ACTION ErrorHandling:
// Alarm_0280	280	Error	Błąd czujnika temperatury zbiornika
// Alarm_0281	281	Error	Błąd grzania zbiornika, brak wzrostu temperatury

IF bAlarmInit THEN
    bAlarmInit := FALSE; 
	fbSourceInfo.Clear();
	fbSourceInfo.sName:=wsLiteral_TO_UTF8(sStationName);//'Machine';
	fbSourceInfo.nId:=iStationIndex;//2700;
	// Alarm_0280	280	Error	Błąd czujnika temperatury zbiornika
    arfbAlarm[0].CreateEx(stEventEntry := TC_EVENTS.AlarmClass.Alarm_0280, bWithConfirmation:= FALSE,  ipSourceInfo:= fbSourceInfo); 
	// Alarm_0281	281	Error	Błąd grzania zbiornika, brak wzrostu temperatury
	arfbAlarm[1].CreateEx(stEventEntry := TC_EVENTS.AlarmClass.Alarm_0281, bWithConfirmation:= FALSE,  ipSourceInfo:= fbSourceInfo);
END_IF
	

//************LISTA BŁĘDÓW***************
bStateError:= (eState=E_Station.eError) OR (eState=E_Station.eResetting) OR bIgnoreError;

IF bEnable THEN
	// Alarm_0280	280	Error	Błąd czujnika temperatury zbiornika
	//Error 1 - Błąd czujnika temperatury zbiornika
	IF (bTemperatureSensorFault OR lrHeaterTemperatureCVSensor = 0 ) THEN
		IF NOT arfbAlarm[0].bActive THEN
			bTempRegulatorReset 	:= TRUE;
			arfbAlarm[0].Raise(nTimeStamp:=0);
		END_IF
	ELSE	
		IF  arfbAlarm[0].bActive AND bReset THEN
			arfbAlarm[0].Clear(nTimeStamp:=0, bResetConfirmation:= FALSE);
		END_IF
// 		bTempRegulatorReset 	:= TRUE;
// 		bError := TRUE;
// 		nErrorNr 				:= 181;
// 		//nErrorNr				:=nErrorNr+iStationIndex;
// 		sErrorDescription 		:= 'Błąd czujnika temperatury zbiornika';	
	END_IF
	// Alarm_0281	281	Error	Błąd grzania zbiornika, brak wzrostu temperatury
	//Error 2 - Błąd czujnika temperatury
	tofbHeaterPWMOut(IN:=bHeaterPWMOut,PT:=T#30S);
	tonHeaterOnAndNotHeating(IN:=tofbHeaterPWMOut.Q AND lrHeaterTemperatureCVSensor=lrHeaterTemperatureCVSensorLast AND NOT bIgnoreError , PT:=T#5M);
	lrHeaterTemperatureCVSensorLast := lrHeaterTemperatureCVSensor;
	IF tonHeaterOnAndNotHeating.Q THEN
		IF NOT arfbAlarm[1].bActive THEN
			bTempRegulatorReset 	:= TRUE;
			arfbAlarm[1].Raise(nTimeStamp:=0);
		END_IF
	ELSE	
		IF  arfbAlarm[1].bActive AND bReset THEN
			arfbAlarm[1].Clear(nTimeStamp:=0, bResetConfirmation:= FALSE);
		END_IF
//  		bTempRegulatorReset 	:= TRUE;
// 		bError := TRUE;
// 		nErrorNr 				:= 182;
// 		//nErrorNr				:=nErrorNr+iStationIndex;
// 		sErrorDescription 		:= 'Błąd grzania zbiornika, brak wzrostu temperatury';	
	END_IF
ELSE
		bError := FALSE;
END_IF
//*******KONIEC LISTA BŁĘDÓW***************

IF bError AND NOT bStateError THEN
	IF eLastState = eRunning THEN
		bCycleNotDone := TRUE;
	END_IF
	eState := E_Station.eError;
END_IF

(*Wyświetlanie błedu na wyjściu*)
bError							:= FALSE;
FOR nAlarmNumerator := 0 TO 19 DO
	bError						:= bError OR arfbAlarm[nAlarmNumerator].bActive;
END_FOR

(*Przepisywanie nazwy stacji*)
sErrorStationName:=WSTRING_TO_STRING(sStationName);
END_ACTION

ACTION HeaterRegulator:
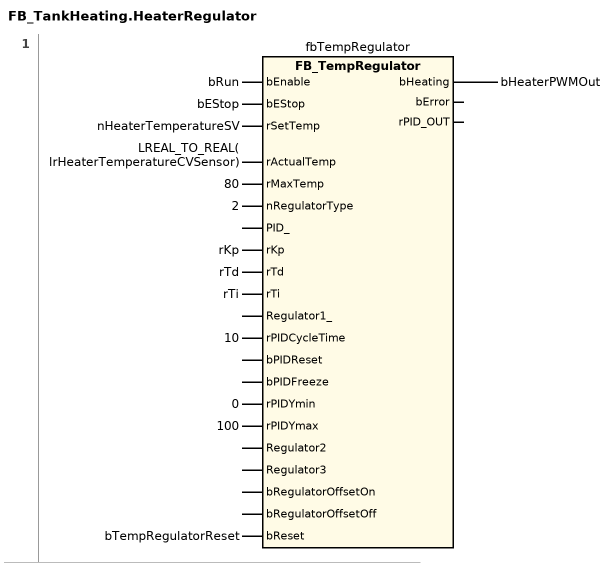
// NETWORK 1
fbTempRegulator(
    bEnable := bRun,
    bEStop := bEStop,
    rSetTemp := nHeaterTemperatureSV,
    rActualTemp := LREAL_TO_REAL(lrHeaterTemperatureCVSensor),
    rMaxTemp := 80,
    nRegulatorType := 2,
    rKp := rKp,
    rTd := rTd,
    rTi := rTi,
    rPIDCycleTime := 10,
    rPIDYmin := 0,
    rPIDYmax := 100,
    bReset := bTempRegulatorReset); // FB_TempRegulator
bHeaterPWMOut := fbTempRegulator.bHeating;
END_ACTION

ACTION Running:

CASE eRunningState OF
	/////////////////////////////	
	E_MassHeatingState.eDisabled:		//Wyłączona
		
		IF bRun THEN
			eRunningState := E_MassHeatingState.eHeating;
		END_IF
		
	/////////////////////////////	
	E_MassHeatingState.eHeating:		//Grzanie
	
		IF (ABS(lrHeaterTemperatureCVSensor-nHeaterTemperatureSV)<nTempHisteresis OR bIgnoreError) THEN
			eRunningState:=E_MassHeatingState.eReady;	
		END_IF
		IF NOT bRun THEN
			eRunningState := E_MassHeatingState.eCooling;
		END_IF
	
	/////////////////////////////	
	E_MassHeatingState.eReady:			//Gotowość
	
		IF (ABS(lrHeaterTemperatureCVSensor-nHeaterTemperatureSV)>nTempHisteresis AND NOT bIgnoreError) THEN
			eRunningState:=E_MassHeatingState.eHeating;
		END_IF
		IF NOT bRun THEN
			eRunningState := E_MassHeatingState.eCooling;
		END_IF
	
	/////////////////////////////	
	E_MassHeatingState.eCooling:		//Chłodzenie
		IF lrHeaterTemperatureCVSensor < 40 THEN
			eRunningState := E_MassHeatingState.eDisabled;
		END_IF
		IF bRun THEN
			eRunningState := E_MassHeatingState.eHeating;
		END_IF

END_CASE
END_ACTION

END_FUNCTION_BLOCK

// ---- POUs/FB/FB_WriteDataToArrayString.TcPOU
FUNCTION_BLOCK FB_WriteDataToArrayString
VAR_INPUT
	bWrite:BOOL;
	nCycleTime:INT;
	lrData1:LREAL;
	lrData2:LREAL;
	lrData2B:LREAL;
	bData3:BOOL;
	bData4:BOOL;
	bData5:BOOL;
	bData2B_ON:BOOL;
END_VAR
VAR_OUTPUT
	AsData:ARRAY [0..500] OF STRING;
END_VAR
VAR
	i: INT;
	sTemp1: STRING;
	sTemp2: STRING;
	sTemp3: STRING;
	sTemp4: STRING;
	sTemp5: STRING;	
	sTemp6: STRING;
	sTemp7: STRING;
	sTemp8: STRING;
	sTemp9: STRING;	
	sTemp10: STRING;	
	sTemp11: STRING;	
	sTemp12: STRING;
	sTemp13: STRING;	
	rtWrite: R_TRIG;
	tonGen1: TON;
	rttonGen1: R_TRIG;
	k: INT;
	tofWrite: TOF;
	fttofWrite: F_TRIG;
	tonWrite: TON;
END_VAR

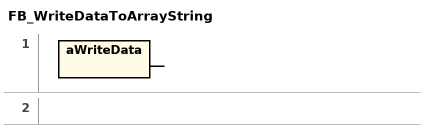
// NETWORK 1
aWriteData();

// NETWORK 2

ACTION aWriteData:
rtWrite(CLK:=bWrite,Q=>);
tofWrite(IN:=bWrite,PT:=T#1S500MS);
tonWrite(IN:=bWrite,PT:=T#100S);
fttofWrite(CLK:=tofWrite.Q,Q=>);
tonWrite.ET;
IF rtWrite.Q THEN
	i:=0;
	//FOR k:=1 TO 500 DO 
	//	AsData[k]:='0;0;0;FALSE;FALSE;FALSE';
	//END_FOR
END_IF

tonGen1(IN:= NOT tonGen1.Q, PT:=INT_TO_TIME(nCycleTime));
rttonGen1(CLK:=tonGen1.Q, Q=>);
	
IF  tofWrite.Q AND rttonGen1.Q THEN
		
	IF i < 500 THEN

		IF NOT bData2B_ON THEN //Bez dodatkowej zmiennej
			//Przygotowanie zmiennej
			//sTemp1:=INT_TO_STRING(i);
			sTemp1:=INT_TO_STRING(TIME_TO_INT(tonWrite.ET)); //Wersja z podawaniem rzeczywistego czasu
			sTemp2:=Concat(sTemp1,';');
			sTemp3:=Concat(sTemp2,INT_TO_STRING(LREAL_TO_INT(lrData1)));
			sTemp4:=Concat(sTemp3,';');	
			sTemp5:=Concat(sTemp4,LREAL_TO_STRING(lrData2));
			sTemp6:=Concat(sTemp5,';');
			sTemp7:=Concat(sTemp6,BOOL_TO_STRING(bData3));
			sTemp8:=Concat(sTemp7,';');		
			sTemp9:=Concat(sTemp8,BOOL_TO_STRING(bData4));
			sTemp10:=Concat(sTemp9,';');
			sTemp11:=Concat(sTemp10,BOOL_TO_STRING(bData5));
			sTemp12:=sTemp11;
			sTemp13:=sTemp12;
		ELSE
			//sTemp1:=INT_TO_STRING(i);
			sTemp1:=INT_TO_STRING(TIME_TO_INT(tonWrite.ET)); //Wersja z podawaniem rzeczywistego czasu
			sTemp2:=Concat(sTemp1,';');
			sTemp3:=Concat(sTemp2,INT_TO_STRING(LREAL_TO_INT(lrData1)));
			sTemp4:=Concat(sTemp3,';');	
			sTemp5:=Concat(sTemp4,LREAL_TO_STRING(lrData2));
			sTemp6:=Concat(sTemp5,';');
			sTemp7:=Concat(sTemp6,LREAL_TO_STRING(lrData2B));
			sTemp8:=Concat(sTemp7,';');		
			sTemp9:=Concat(sTemp8,BOOL_TO_STRING(bData3));
			sTemp10:=Concat(sTemp9,';');		
			sTemp11:=Concat(sTemp10,BOOL_TO_STRING(bData4));
			sTemp12:=Concat(sTemp11,';');
			sTemp13:=Concat(sTemp12,BOOL_TO_STRING(bData5));
		END_IF
		
		
		//Wpisanie zmiennej do tablicy
		AsData[i]:=sTemp13;
		
		i:=i+1;
		
	END_IF
END_IF	
IF fttofWrite.Q THEN
	IF NOT bData2B_ON THEN //Bez dodatkowej zmiennej
			FOR k:=i TO 500 DO 
			  AsData[k]:='0;0;0;FALSE;FALSE;FALSE';
			END_FOR
	ELSE
			FOR k:=i TO 500 DO 
			  AsData[k]:='0;0;0;0;FALSE;FALSE;FALSE';
			END_FOR
	END_IF
END_IF
END_ACTION

END_FUNCTION_BLOCK

// ---- POUs/FB/FB_WriteDataToArrayOfArrays.TcPOU
FUNCTION_BLOCK FB_WriteDataToArrayOfArrays
VAR_INPUT
	bWrite			:BOOL;
	udiCycleTime	:UDINT;
	lrAiData0		:LREAL;
	lrAiData1		:LREAL;
	lrAiData2		:LREAL;
	lrAiData3		:LREAL;
	lrAiData4		:LREAL;	
END_VAR
VAR_OUTPUT
	AiData			:ARRAY [0..5,0..500] OF INT;	
END_VAR
VAR
	i,j				:INT;	
	rtWrite			:R_TRIG;
	tonGen1			:TON;
	rttonGen1		:R_TRIG;
	k				:INT;
	tofWrite		:TOF;
	fttofWrite		:F_TRIG;
	tonWrite		:TON;
END_VAR

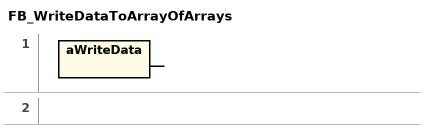
// NETWORK 1
aWriteData();

// NETWORK 2

ACTION aWriteData:
rtWrite		(CLK	:=	bWrite,Q=>);
tofWrite	(IN		:=	bWrite,PT:=T#1S500MS);
tonWrite	(IN		:=	bWrite,PT:=T#100S);
fttofWrite	(CLK	:=	tofWrite.Q,Q=>);
tonWrite.ET;
IF rtWrite.Q THEN
	i:=0;
END_IF

tonGen1(IN:= NOT tonGen1.Q, PT:=T#10MS);
rttonGen1(CLK:=tonGen1.Q, Q=>);
	
IF  tofWrite.Q AND rttonGen1.Q THEN
		
	IF i < 500 THEN	
		AiData[0,i]	:=	LREAL_TO_INT(lrAiData0);	
		AiData[1,i]	:=	LREAL_TO_INT(lrAiData1);		
		AiData[2,i]	:=	LREAL_TO_INT(lrAiData2);	
		AiData[3,i]	:=	LREAL_TO_INT(lrAiData3);		
		AiData[4,i]	:=	LREAL_TO_INT(lrAiData4);		
		i:=i+1;	
	
	END_IF
END_IF	
IF fttofWrite.Q THEN
	FOR k:=i TO 500 DO 
		//AstData[k].udiCycleTime :=	udiCycleTime;
		AiData[0,i]	:=	0;	
		AiData[1,i]	:=	0;		
		AiData[2,i]	:=	0;	
		AiData[3,i]	:=	0;	
		AiData[4,i]	:=	0;		
	END_FOR
	AiData[4,500] :=	UDINT_TO_INT(udiCycleTime);
END_IF
END_ACTION

END_FUNCTION_BLOCK

// ---- POUs/FB/Blinkers/FB_Blink_AS.TcPOU
(********************************************************************************************)
(*							Beckhoff Automation Poland										*)
(*								FB_Blink_AS	 v1.1											*)
(*									9.11.2007												*)
(*						Blok funkcyjny zegara asynchronicznego								*)
(*__________________________________________________________________________________________*)

FUNCTION_BLOCK FB_Blink_AS
VAR_INPUT
	T1										:	TIME;				(*Czas, gdy wyjście przyjmuje wartość TRUE*)
	T0										:	TIME;				(*Czas, gdy wyjście przyjmuje wartość FALSE*)
END_VAR
VAR_OUTPUT
	Q										:	BOOL;				(*Wyjscie*)
END_VAR
VAR
	ton1									:	TON;
	ton2									:	TON;
END_VAR

ton1(IN:= NOT ton2.Q, PT:=T0);
Q:=ton1.Q;
ton2(IN:=ton1.Q , PT:=T1);

END_FUNCTION_BLOCK

// ---- POUs/FB/Various/FB_FilterEx.TcPOU
//==================================================================================================
//							Beckhoff Automation Poland
//									23.11.2016
//			Bloczek do filtru inercyjnego do wygladzania przebiegow,					
//					czas próbkowania wyliczany wewnętrznie
//  v1.1	|| TC v 3.1.4020.28		|| - poprawienie inicjalizacji, notacja wegierska
// 	v1.0	|| TC v 3.1.4020.0		|| - pierwsza wersja
//==================================================================================================
FUNCTION_BLOCK FB_FilterEx
VAR_INPUT
	rIn										: REAL;					// Sygnal wejsciowy
	tTimeConstant							: TIME;					// Stala czasowa T gdy rOut = 0,63 * rIn 
END_VAR
VAR_OUTPUT
	rOut									: REAL;					// Przefiltrowany sygnal wyjsciowy, 
END_VAR
VAR
	rLastOut								: REAL;					// Wartosc wyjscia w poprzednim cyklu
	rCycleTime								: REAL; 				// [ms]
	rTimeConst								: REAL;					// [ms]
	tX										: TIME;					// Aktualny czas
	tY 										: TIME;					// Zmienna pomocnicza, poprzedni czas
	tCycleTime								: TIME;					// Wyliczony czas cyklu
	bFirstCycle								: BOOL := TRUE;			// Flaga pierwszego cyklu - nie mamy jeszce wyliczonego prawidlowo czasu cylu 
																	// - potrzebujemy dwoch cylki do odjecia czasu
END_VAR

// Obliczenie czasu cyklu do inkrementu
tX 					:= TIME();
IF NOT bFirstCycle THEN
	tCycleTime 		:= tX - tY;
END_IF
tY 					:= tX;
// Przeliczenie czasu na typ REAL
rCycleTime 			:= TIME_TO_REAL(tCycleTime);
rTimeConst 			:= TIME_TO_REAL(tTimeConstant);
// Wyliczenie wyjscia tylko jesli stala czasowa wieksza od 1 ms i zakonczylismy inicjalizacje
IF NOT bFirstCycle AND rTimeConst > 0.001 THEN
	rOut 			:= rLastOut + (rIn - rLastOut) * rCycleTime/rTimeConst;
	rLastOut 		:= rOut;
END_IF
// Zerowanie flagu pierwszego cyklu
bFirstCycle 		:= FALSE;

END_FUNCTION_BLOCK

// ---- POUs/FB/Various/F_Scaling.TcPOU
(************************************************************************************)
(*							Beckhoff Automation Poland								*)
(*								F_Scaling v2										*)
(*									3.11.2011										*)
(*					Funkcja skalująca wartość wejściową rValue na wyjściową 		*)
(*__________________________________________________________________________________*)
FUNCTION F_Scaling: DINT
VAR_INPUT
	rValue	:	DINT;	(*Zmienna skalowana*)
	rXmin	:	DINT;	(*Dolny zakres zmiennej przeskalowanej*)
	rXmax	:	DINT;	(*Górny zakres zmiennej przeskalowanej*)
	rYmin	:	DINT;	(*Dolny zakres zmiennej skalowanej*)
	rYmax	:	DINT;	(*Górny zakres zmiennej skalowanej*)
END_VAR
VAR
	rfA		:	DINT;	(*Wspólczynnik kierunkowy prostej*)
	rfB		:	DINT;	(*Współczynnik przesunięcia prostej*)
END_VAR

IF (rValue > rXmax) THEN
	F_Scaling := rYmax;
ELSIF (rValue <= rXmin) THEN
	F_Scaling := rYmin;
ELSE
	IF (((rXmax - rXmin) < 0.01) AND ((rXmax - rXmin) > -0.01)) THEN
		F_Scaling := rYmin;
	ELSE
		rfA := (rYmax - rYmin) / (rXmax - rXmin);
		rfB := rYmax - rfA * rXmax;
		F_Scaling := rfA * rValue + rfB;
	END_IF;
END_IF

END_FUNCTION

// ---- POUs/P02_DispencersCharts.TcPOU
PROGRAM P02_DispencersCharts
VAR
	tonDispencer1SuckingValveOpenedSensor				:	TON;			//Symulacja czujników 
	tonDispencer1DosingValveOpenedSensor				:	TON;			//Symulacja czujników 
	tonDispencer1DosingValveClosedSensor				:	TON;			//Symulacja czujników 
	tonDispencer1SuckingValveClosedSensor				: 	TON;
	
	QbDispencer1SuckingValveActuator					:	BOOL;
	QbDispencer1DosingValveActuator 					:	BOOL;
	
	fbDisp												:	FB_ServoDispencerServoLifter;
	iVirtualCycleCase									:	INT;
	
	bRun												:	BOOL;
	
	bManualMovement           							:	BOOL;  //Zezwolenie na ruchy ręczne
	bManualSync				  							:	BOOL;	// Synchronizacja-Przejazd tłoka i podnośnika do określonej pozycji
    lrManualOverride          							:	LREAL; //Procentowa redukcja prędkości wszystkich serw (Tylko w trybie serwisowym)
    bManualPullingFast        							:	BOOL;  //Przeciąganie dozownika szybkie
    bManualPullingSlow        							:	BOOL;  //Przeciąganie dozownika wolne
	bManualCleaningMode		  							:	BOOL;	//Włączenie trybu mycia
	bManualCleaning			  							:	BOOL;	//Włącz mycie, do synchronizacji
    bManualPistonBack         							:	BOOL;  //Ruch ręczny podnośnikiem stacji w górę
    bManualPistonForward      							:	BOOL;  //Ruch ręczny podnośnikiem stacji w dół
    bManualSuckingValve       							:	BOOL;  //Otwarcie ręczne zaworu ssącego
    bManualDosingValve        							:	BOOL;  //Otwarcie ręczne zaworu dozującego (iglicy)
    bManualDropCatcherForward 							:	BOOL;  //Wysunięcie ręczne tacki kropel
    bManualLifterUp           							:	BOOL;  //Podniesienie ręczne stacji dozownika (podpinać zmienną jeśli bDispencerWithLifter=TRUE)
    bManualLifterDown         							:	BOOL;  //Opuszczenie ręczne stacji dozownika (podpinać zmienną jeśli bDispencerWithLifter=TRUE)
	
	DispencerAxisRef       								: 	AXIS_REF; //Struktura sterowania NC dla serwa Dozownika
    DispencerLifterAxisRef 								: 	AXIS_REF;
	
	//lrDispencer1DoseVolumeShow							: 	LREAL	:=495;
	//lrDispencer1Phase1VolumeShow						: 	LREAL	:=0;
	//lrDispencer1Phase2VolumeShow						: 	LREAL	:=00;
	//lrDispencer1Phase1VelocityShow						: 	LREAL	:=140;
	//lrDispencer1Phase2VelocityShow						: 	LREAL	:=140;
	//lrDispencer1Phase3VelocityShow						: 	LREAL	:=50;
	//lrDispencer1SuckVelocityShow						: 	LREAL	:=300;
	//lrDispencer1Phase1AccelerationShow					: 	LREAL	:=600;
	//lrDispencer1Phase2AccelerationShow					: 	LREAL	:=400;
	//lrDispencer1Phase3AccelerationShow					: 	LREAL	:=50;
	//lrDispencer1SuckAccelerationShow					: 	LREAL	:=3000;
	//lrDispencer1Phase1DecelerationShow					: 	LREAL	:=150;
	//lrDispencer1Phase2DecelerationShow					: 	LREAL	:=2000;
	//lrDispencer1Phase3DecelerationShow					: 	LREAL	:=50;
	//udiDispencer1DosingDoneDelayTimeShow				: 	UDINT	:=10;
	//lrDispencer1SuckValveOpenVolumeShow					: 	LREAL	:=0;
	//lrDispencer1SuckValveOpenTimeDelayShow				: 	LREAL	:=0;
	//lrDispencer1SuckValveCloseVolumeShow				: 	LREAL	:=0;
	//lrDispencer1SuckValveCloseTimeDelayShow				: 	LREAL	:=0;
	//lrDispencer1DoseValveOpenVolumeShow					: 	LREAL	:=0;
	//lrDispencer1DoseValveOpenTimeAccShow				: 	LREAL	:=200;
	//lrDispencer1DoseValveCloseVolumeShow				: 	LREAL	:=1;
	//lrDispencer1DoseValveCloseTimeDecShow				: 	LREAL	:=0;
	//lrDispencer1DoseSuckingVolumeShow					: 	LREAL	:=0;
	//lrDispencer1DoseSuckingTimeDelayShow				: 	LREAL	:=0;
	//bDispencer1DoseSuckingShow							: 	BOOL 	:=FALSE;
	//bDispencer1LiftSynchroPh1Show						: 	BOOL 	:=FALSE;
	//bDispencer1LiftSynchroPh2Show						: 	BOOL 	:=TRUE;
	//bDispencer1LiftSynchroPh3Show						: 	BOOL 	:=TRUE;
	//lrDispencer1LifterStartDosePositionShow				: 	LREAL 	:=80;
	//lrDispencer1LifterStopDosePositionShow				: 	LREAL 	:=192;
	//lrDispencer1LifterVelocityShow						: 	LREAL 	:=1050;
	//lrDispencer1LifterAccelerationShow					: 	LREAL 	:=15000;
	//lrDispencer1LifterDecelerationShow					: 	LREAL 	:=15000;
	//
	//lrDispencersCatchHeightSVShow						:	LREAL	:=86;  				// Pozycja chwytaka
	//lrDispencersLifterReadyPosition						: 	LREAL	:=	270;
	
	bServiceBrakeOff									:	BOOL;
	
	
	rt_DrawChart										:	R_TRIG;
	tonChartRun											:	ton;
	
	fbChart0											:	FB_ChartGenerator;
	aPoints0											:	ARRAY [0..11,0..599] OF ST_Point;	// Sam wykres wybrando doziwniki + jego simulacji
	
	fbChart1											:	FB_ChartGenerator;
	aPoints1											:	ARRAY [0..11,0..599] OF ST_Point;	// Sam wykres wybrando doziwniki + jego simulacji

	fbChart2											:	FB_ChartGenerator;
	aPoints2											:	ARRAY [0..11,0..599] OF ST_Point;	// Sam wykres wybrando doziwniki + jego simulacji

	fbChart3											:	FB_ChartGenerator;
	aPoints3											:	ARRAY [0..11,0..599] OF ST_Point;	// Sam wykres wybrando doziwniki + jego simulacji

		tDelayDispencerValve								: TIME;
	
END_VAR
VAR_INPUT
	bDispencersSyncSim: BOOL;
END_VAR
VAR_OUTPUT
	bDispenserSimMultiMasterSyncOut:BOOL;
END_VAR

tDelayDispencerValve																			:= T#50MS;
tonDispencer1SuckingValveClosedSensor(IN:=NOT QbDispencer1SuckingValveActuator, PT:=tDelayDispencerValve);
tonDispencer1SuckingValveOpenedSensor(IN:=QbDispencer1SuckingValveActuator,PT:=tDelayDispencerValve);
tonDispencer1DosingValveOpenedSensor(IN:=QbDispencer1DosingValveActuator ,PT:=tDelayDispencerValve);
tonDispencer1DosingValveClosedSensor(IN:=NOT QbDispencer1DosingValveActuator ,PT:=tDelayDispencerValve);

ACT_SimDispencer();
ACT_VirtualCycle();
ACT_ChartDrawers();

IF VIS.udiDossagerNum = 0 THEN
	VIS.nDrawLenght:= fbChart0.nTimeMarkerEnd+500;
ELSIF VIS.udiDossagerNum = 1 THEN
	VIS.nDrawLenght:= fbChart1.nTimeMarkerEnd+500;
ELSIF VIS.udiDossagerNum = 2 THEN
	VIS.nDrawLenght:= fbChart2.nTimeMarkerEnd+500;
ELSIF VIS.udiDossagerNum = 3 THEN
	VIS.nDrawLenght:= fbChart3.nTimeMarkerEnd+500;
END_IF

ACTION ACT_ChartDrawers:
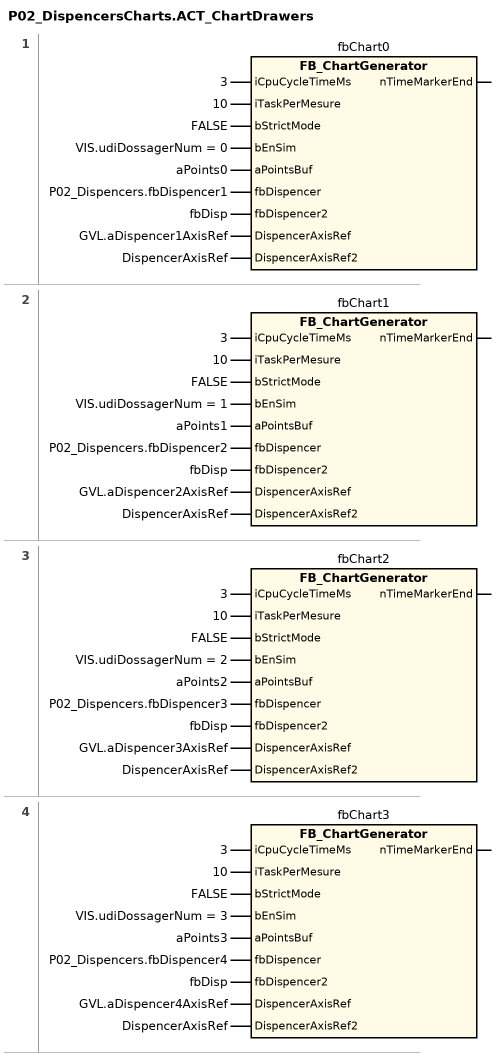
// NETWORK 1
fbChart0(
    iCpuCycleTimeMs := 3,
    iTaskPerMesure := 10,
    bStrictMode := FALSE,
    bEnSim := VIS.udiDossagerNum = 0,
    aPointsBuf := aPoints0,
    fbDispencer := P02_Dispencers.fbDispencer1,
    fbDispencer2 := fbDisp,
    DispencerAxisRef := GVL.aDispencer1AxisRef,
    DispencerAxisRef2 := DispencerAxisRef); // FB_ChartGenerator

// NETWORK 2
fbChart1(
    iCpuCycleTimeMs := 3,
    iTaskPerMesure := 10,
    bStrictMode := FALSE,
    bEnSim := VIS.udiDossagerNum = 1,
    aPointsBuf := aPoints1,
    fbDispencer := P02_Dispencers.fbDispencer2,
    fbDispencer2 := fbDisp,
    DispencerAxisRef := GVL.aDispencer2AxisRef,
    DispencerAxisRef2 := DispencerAxisRef); // FB_ChartGenerator

// NETWORK 3
fbChart2(
    iCpuCycleTimeMs := 3,
    iTaskPerMesure := 10,
    bStrictMode := FALSE,
    bEnSim := VIS.udiDossagerNum = 2,
    aPointsBuf := aPoints2,
    fbDispencer := P02_Dispencers.fbDispencer3,
    fbDispencer2 := fbDisp,
    DispencerAxisRef := GVL.aDispencer3AxisRef,
    DispencerAxisRef2 := DispencerAxisRef); // FB_ChartGenerator

// NETWORK 4
fbChart3(
    iCpuCycleTimeMs := 3,
    iTaskPerMesure := 10,
    bStrictMode := FALSE,
    bEnSim := VIS.udiDossagerNum = 3,
    aPointsBuf := aPoints3,
    fbDispencer := P02_Dispencers.fbDispencer4,
    fbDispencer2 := fbDisp,
    DispencerAxisRef := GVL.aDispencer4AxisRef,
    DispencerAxisRef2 := DispencerAxisRef); // FB_ChartGenerator
END_ACTION

ACTION ACT_SimDispencer:
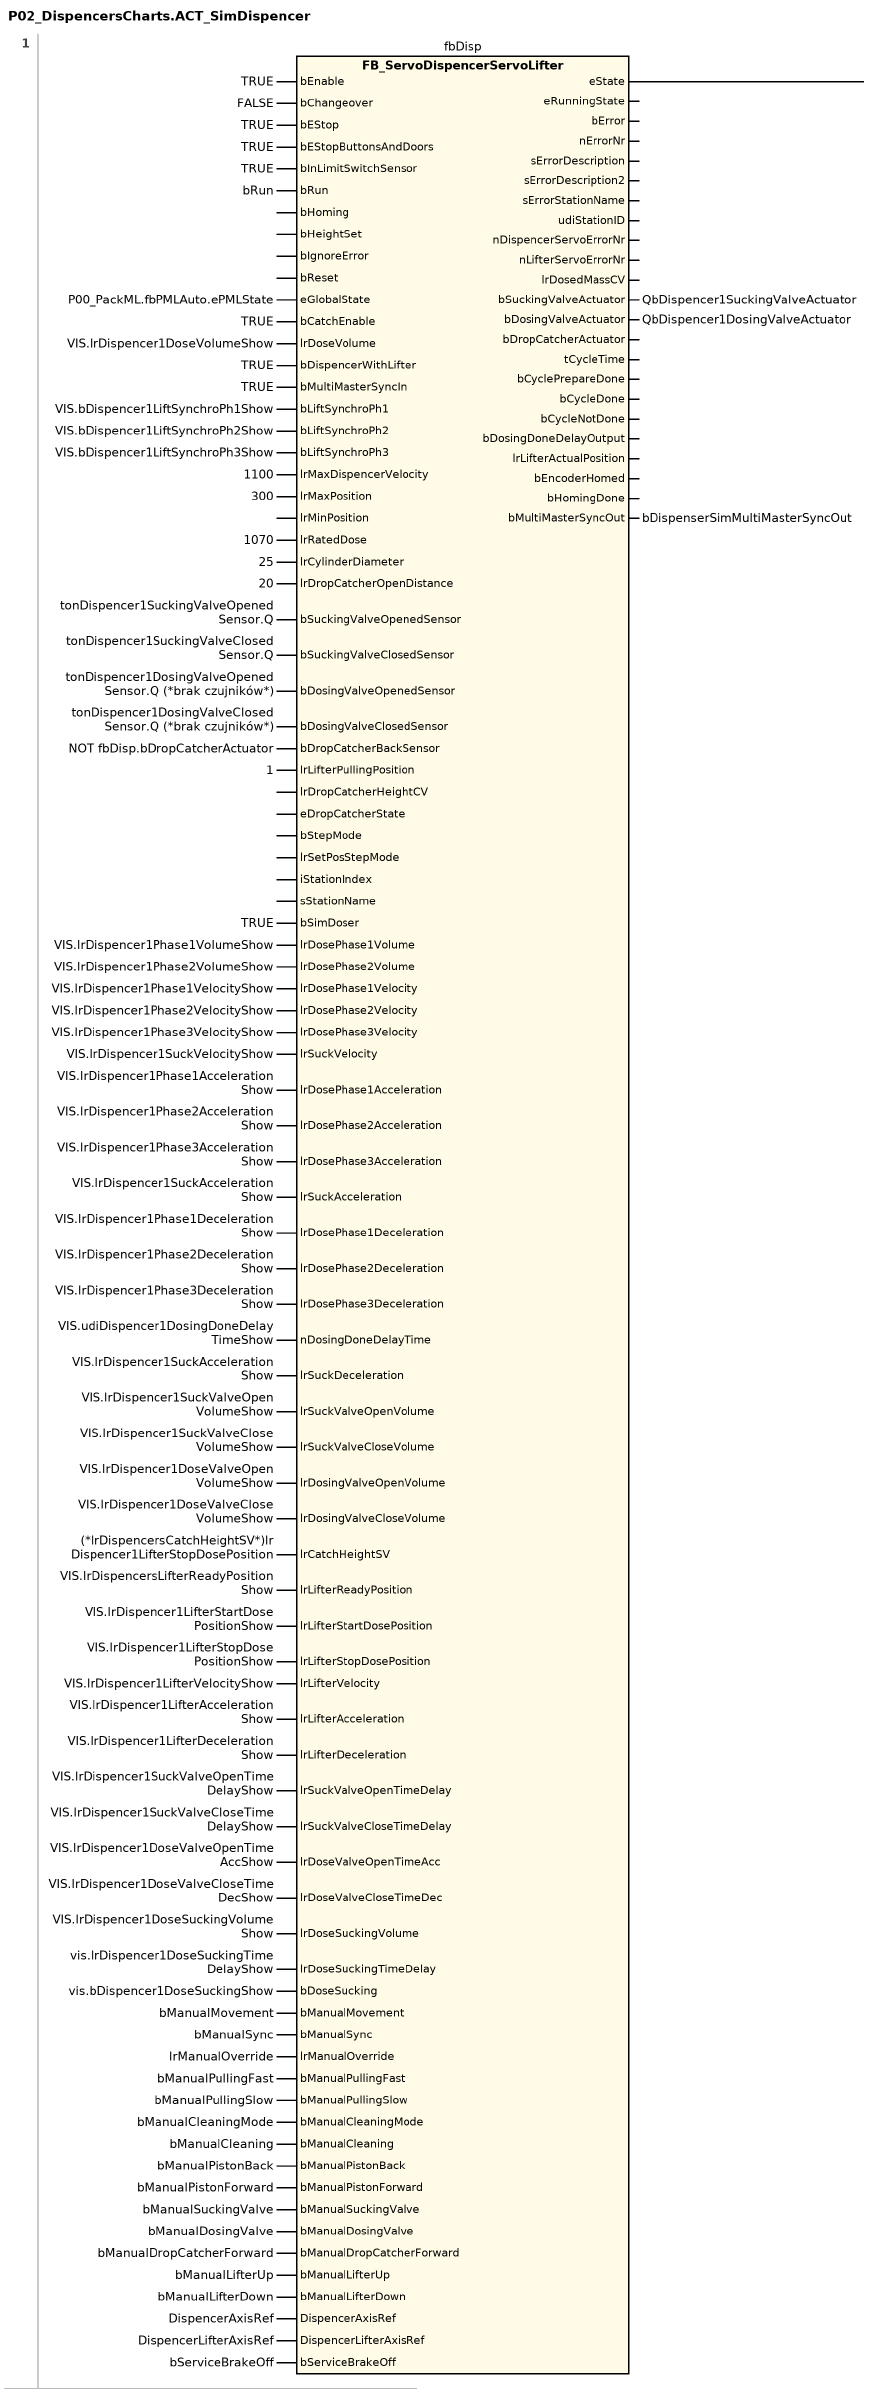
// NETWORK 1
fbDisp(
    bEnable := TRUE,
    bChangeover := FALSE,
    bEStop := TRUE,
    bEStopButtonsAndDoors := TRUE,
    bInLimitSwitchSensor := TRUE,
    bRun := bRun,
    eGlobalState := P00_PackML.fbPMLAuto.ePMLState,
    bCatchEnable := TRUE,
    lrDoseVolume := VIS.lrDispencer1DoseVolumeShow,
    bDispencerWithLifter := TRUE,
    bMultiMasterSyncIn := TRUE,
    bLiftSynchroPh1 := VIS.bDispencer1LiftSynchroPh1Show,
    bLiftSynchroPh2 := VIS.bDispencer1LiftSynchroPh2Show,
    bLiftSynchroPh3 := VIS.bDispencer1LiftSynchroPh3Show,
    lrMaxDispencerVelocity := 1100,
    lrMaxPosition := 300,
    lrRatedDose := 1070,
    lrCylinderDiameter := 25,
    lrDropCatcherOpenDistance := 20,
    bSuckingValveOpenedSensor := tonDispencer1SuckingValveOpenedSensor.Q,
    bSuckingValveClosedSensor := tonDispencer1SuckingValveClosedSensor.Q,
    bDosingValveOpenedSensor := tonDispencer1DosingValveOpenedSensor.Q (*brak czujników*),
    bDosingValveClosedSensor := tonDispencer1DosingValveClosedSensor.Q (*brak czujników*),
    bDropCatcherBackSensor := NOT fbDisp.bDropCatcherActuator,
    lrLifterPullingPosition := 1,
    bSimDoser := TRUE,
    lrDosePhase1Volume := VIS.lrDispencer1Phase1VolumeShow,
    lrDosePhase2Volume := VIS.lrDispencer1Phase2VolumeShow,
    lrDosePhase1Velocity := VIS.lrDispencer1Phase1VelocityShow,
    lrDosePhase2Velocity := VIS.lrDispencer1Phase2VelocityShow,
    lrDosePhase3Velocity := VIS.lrDispencer1Phase3VelocityShow,
    lrSuckVelocity := VIS.lrDispencer1SuckVelocityShow,
    lrDosePhase1Acceleration := VIS.lrDispencer1Phase1AccelerationShow,
    lrDosePhase2Acceleration := VIS.lrDispencer1Phase2AccelerationShow,
    lrDosePhase3Acceleration := VIS.lrDispencer1Phase3AccelerationShow,
    lrSuckAcceleration := VIS.lrDispencer1SuckAccelerationShow,
    lrDosePhase1Deceleration := VIS.lrDispencer1Phase1DecelerationShow,
    lrDosePhase2Deceleration := VIS.lrDispencer1Phase2DecelerationShow,
    lrDosePhase3Deceleration := VIS.lrDispencer1Phase3DecelerationShow,
    nDosingDoneDelayTime := VIS.udiDispencer1DosingDoneDelayTimeShow,
    lrSuckDeceleration := VIS.lrDispencer1SuckAccelerationShow,
    lrSuckValveOpenVolume := VIS.lrDispencer1SuckValveOpenVolumeShow,
    lrSuckValveCloseVolume := VIS.lrDispencer1SuckValveCloseVolumeShow,
    lrDosingValveOpenVolume := VIS.lrDispencer1DoseValveOpenVolumeShow,
    lrDosingValveCloseVolume := VIS.lrDispencer1DoseValveCloseVolumeShow,
    lrCatchHeightSV := (*lrDispencersCatchHeightSV*)lrDispencer1LifterStopDosePosition,
    lrLifterReadyPosition := VIS.lrDispencersLifterReadyPositionShow,
    lrLifterStartDosePosition := VIS.lrDispencer1LifterStartDosePositionShow,
    lrLifterStopDosePosition := VIS.lrDispencer1LifterStopDosePositionShow,
    lrLifterVelocity := VIS.lrDispencer1LifterVelocityShow,
    lrLifterAcceleration := VIS.lrDispencer1LifterAccelerationShow,
    lrLifterDeceleration := VIS.lrDispencer1LifterDecelerationShow,
    lrSuckValveOpenTimeDelay := VIS.lrDispencer1SuckValveOpenTimeDelayShow,
    lrSuckValveCloseTimeDelay := VIS.lrDispencer1SuckValveCloseTimeDelayShow,
    lrDoseValveOpenTimeAcc := VIS.lrDispencer1DoseValveOpenTimeAccShow,
    lrDoseValveCloseTimeDec := VIS.lrDispencer1DoseValveCloseTimeDecShow,
    lrDoseSuckingVolume := VIS.lrDispencer1DoseSuckingVolumeShow,
    lrDoseSuckingTimeDelay := vis.lrDispencer1DoseSuckingTimeDelayShow,
    bDoseSucking := vis.bDispencer1DoseSuckingShow,
    bManualMovement := bManualMovement,
    bManualSync := bManualSync,
    lrManualOverride := lrManualOverride,
    bManualPullingFast := bManualPullingFast,
    bManualPullingSlow := bManualPullingSlow,
    bManualCleaningMode := bManualCleaningMode,
    bManualCleaning := bManualCleaning,
    bManualPistonBack := bManualPistonBack,
    bManualPistonForward := bManualPistonForward,
    bManualSuckingValve := bManualSuckingValve,
    bManualDosingValve := bManualDosingValve,
    bManualDropCatcherForward := bManualDropCatcherForward,
    bManualLifterUp := bManualLifterUp,
    bManualLifterDown := bManualLifterDown,
    DispencerAxisRef := DispencerAxisRef,
    DispencerLifterAxisRef := DispencerLifterAxisRef,
    bServiceBrakeOff := bServiceBrakeOff,
    bSuckingValveActuator => QbDispencer1SuckingValveActuator,
    bDosingValveActuator => QbDispencer1DosingValveActuator,
    bMultiMasterSyncOut => bDispenserSimMultiMasterSyncOut); // FB_ServoDispencerServoLifter
END_ACTION

ACTION ACT_VirtualCycle:
rt_DrawChart		(	CLK	:=	VIS.bDrawChart						);
tonChartRun			(	IN	:=	iVirtualCycleCase = 100,	PT	:=	T#15S	);

CASE iVirtualCycleCase OF
	0:
		IF (rt_DrawChart.Q) THEN
			CASE VIS.udiDossagerNum OF
				0,1:
					iVirtualCycleCase						:=	10;
				2,3:
					iVirtualCycleCase						:=	20;
			END_CASE
		END_IF
	10:
		//Copy parameters from RECIPE to FB
		//lrDispencer1DoseVolumeShow							:=    VIS.lrDispencer1DoseVolumeShow				;
		//lrDispencer1Phase1VolumeShow						:=    VIS.lrDispencer1Phase1VolumeShow				;
		//lrDispencer1Phase2VolumeShow						:=    VIS.lrDispencer1Phase2VolumeShow				;
		//lrDispencer1Phase1VelocityShow						:=    VIS.lrDispencer1Phase1VelocityShow			;
		//lrDispencer1Phase2VelocityShow						:=    VIS.lrDispencer1Phase2VelocityShow			;
		//lrDispencer1Phase3VelocityShow						:=    VIS.lrDispencer1Phase3VelocityShow			;
		//lrDispencer1SuckVelocityShow						:=    VIS.lrDispencer1SuckVelocityShow				;
		//lrDispencer1Phase1AccelerationShow					:=    VIS.lrDispencer1Phase1AccelerationShow		;
		//lrDispencer1Phase2AccelerationShow					:=    VIS.lrDispencer1Phase2AccelerationShow		;
		//lrDispencer1Phase3AccelerationShow					:=    VIS.lrDispencer1Phase3AccelerationShow		;
		//lrDispencer1SuckAccelerationShow					:=    VIS.lrDispencer1SuckAccelerationShow			;
		//lrDispencer1Phase1DecelerationShow					:=    VIS.lrDispencer1Phase1DecelerationShow		;
		//lrDispencer1Phase2DecelerationShow					:=    VIS.lrDispencer1Phase2DecelerationShow		;
		//lrDispencer1Phase3DecelerationShow					:=    VIS.lrDispencer1Phase3DecelerationShow		;
		//udiDispencer1DosingDoneDelayTimeShow				:=    VIS.udiDispencer1DosingDoneDelayTimeShow		;
		//lrDispencer1SuckValveOpenVolumeShow					:=    VIS.lrDispencer1SuckValveOpenVolumeShow		;
		//lrDispencer1SuckValveOpenTimeDelayShow				:=    VIS.lrDispencer1SuckValveOpenTimeDelayShow	;
		//lrDispencer1SuckValveCloseVolumeShow				:=    VIS.lrDispencer1SuckValveCloseVolumeShow		;
		//lrDispencer1SuckValveCloseTimeDelayShow				:=    VIS.lrDispencer1SuckValveCloseTimeDelayShow	;
		//lrDispencer1DoseValveOpenVolumeShow					:=    VIS.lrDispencer1DoseValveOpenVolumeShow		;
		//lrDispencer1DoseValveOpenTimeAccShow				:=    VIS.lrDispencer1DoseValveOpenTimeAccShow		;
		//lrDispencer1DoseValveCloseVolumeShow				:=    VIS.lrDispencer1DoseValveCloseVolumeShow		;
		//lrDispencer1DoseValveCloseTimeDecShow				:=    VIS.lrDispencer1DoseValveCloseTimeDecShow		;
		//lrDispencer1DoseSuckingVolumeShow					:=    VIS.lrDispencer1DoseSuckingVolumeShow			;
		//lrDispencer1DoseSuckingTimeDelayShow				:=    VIS.lrDispencer1DoseSuckingTimeDelayShow		;
		//bDispencer1DoseSuckingShow							:=    VIS.bDispencer1DoseSuckingShow				;
		//bDispencer1LiftSynchroPh1Show						:=    VIS.bDispencer1LiftSynchroPh1Show				;
		//bDispencer1LiftSynchroPh2Show						:=    VIS.bDispencer1LiftSynchroPh2Show				;
		//bDispencer1LiftSynchroPh3Show						:=    VIS.bDispencer1LiftSynchroPh3Show				;
		//lrDispencer1LifterStartDosePositionShow				:=    VIS.lrDispencer1LifterStartDosePositionShow	;
		//lrDispencer1LifterStopDosePositionShow				:=    VIS.lrDispencer1LifterStopDosePositionShow	;
		//lrDispencer1LifterVelocityShow						:=    VIS.lrDispencer1LifterVelocityShow			;
		//lrDispencer1LifterAccelerationShow					:=    VIS.lrDispencer1LifterAccelerationShow		;
		//lrDispencer1LifterDecelerationShow					:=    VIS.lrDispencer1LifterDecelerationShow		;
		//                                                  
		//lrDispencersCatchHeightSVShow						:=    VIS.lrDispencersCatchHeightSVShow				;  	// Pozycja chwytaka
		//lrDispencersLifterReadyPosition						:=    VIS.lrDispencersLifterReadyPositionShow		;
		
		iVirtualCycleCase									:=	 100;
	20:
		//Copy parameters from RECIPE to FB
		//lrDispencer1DoseVolumeShow							:=    VIS.lrDispencer2DoseVolumeShow				;
		//lrDispencer1Phase1VolumeShow						:=    VIS.lrDispencer2Phase1VolumeShow				;
		//lrDispencer1Phase2VolumeShow						:=    VIS.lrDispencer2Phase2VolumeShow				;
		//lrDispencer1Phase1VelocityShow						:=    VIS.lrDispencer2Phase1VelocityShow			;
		//lrDispencer1Phase2VelocityShow						:=    VIS.lrDispencer2Phase2VelocityShow			;
		//lrDispencer1Phase3VelocityShow						:=    VIS.lrDispencer2Phase3VelocityShow			;
		//lrDispencer1SuckVelocityShow						:=    VIS.lrDispencer2SuckVelocityShow				;
		//lrDispencer1Phase1AccelerationShow					:=    VIS.lrDispencer2Phase1AccelerationShow		;
		//lrDispencer1Phase2AccelerationShow					:=    VIS.lrDispencer2Phase2AccelerationShow		;
		//lrDispencer1Phase3AccelerationShow					:=    VIS.lrDispencer2Phase3AccelerationShow		;
		//lrDispencer1SuckAccelerationShow					:=    VIS.lrDispencer2SuckAccelerationShow			;
		//lrDispencer1Phase1DecelerationShow					:=    VIS.lrDispencer2Phase1DecelerationShow		;
		//lrDispencer1Phase2DecelerationShow					:=    VIS.lrDispencer2Phase2DecelerationShow		;
		//lrDispencer1Phase3DecelerationShow					:=    VIS.lrDispencer2Phase3DecelerationShow		;
		//udiDispencer1DosingDoneDelayTimeShow				:=    VIS.udiDispencer2DosingDoneDelayTimeShow		;
		//lrDispencer1SuckValveOpenVolumeShow					:=    VIS.lrDispencer2SuckValveOpenVolumeShow		;
		//lrDispencer1SuckValveOpenTimeDelayShow				:=    VIS.lrDispencer2SuckValveOpenTimeDelayShow	;
		//lrDispencer1SuckValveCloseVolumeShow				:=    VIS.lrDispencer2SuckValveCloseVolumeShow		;
		//lrDispencer1SuckValveCloseTimeDelayShow				:=    VIS.lrDispencer2SuckValveCloseTimeDelayShow	;
		//lrDispencer1DoseValveOpenVolumeShow					:=    VIS.lrDispencer2DoseValveOpenVolumeShow		;
		//lrDispencer1DoseValveOpenTimeAccShow				:=    VIS.lrDispencer2DoseValveOpenTimeAccShow		;
		//lrDispencer1DoseValveCloseVolumeShow				:=    VIS.lrDispencer2DoseValveCloseVolumeShow		;
		//lrDispencer1DoseValveCloseTimeDecShow				:=    VIS.lrDispencer2DoseValveCloseTimeDecShow		;
		//lrDispencer1DoseSuckingVolumeShow					:=    VIS.lrDispencer2DoseSuckingVolumeShow			;
		//lrDispencer1DoseSuckingTimeDelayShow				:=    VIS.lrDispencer2DoseSuckingTimeDelayShow		;
		//bDispencer1DoseSuckingShow							:=    VIS.bDispencer2DoseSuckingShow				;
		//bDispencer1LiftSynchroPh1Show						:=    VIS.bDispencer2LiftSynchroPh1Show				;
		//bDispencer1LiftSynchroPh2Show						:=    VIS.bDispencer2LiftSynchroPh2Show				;
		//bDispencer1LiftSynchroPh3Show						:=    VIS.bDispencer2LiftSynchroPh3Show				;
		//lrDispencer1LifterStartDosePositionShow				:=    VIS.lrDispencer2LifterStartDosePositionShow	;
		//lrDispencer1LifterStopDosePositionShow				:=    VIS.lrDispencer2LifterStopDosePositionShow	;
		//lrDispencer1LifterVelocityShow						:=    VIS.lrDispencer2LifterVelocityShow			;
		//lrDispencer1LifterAccelerationShow					:=    VIS.lrDispencer2LifterAccelerationShow		;
		//lrDispencer1LifterDecelerationShow					:=    VIS.lrDispencer2LifterDecelerationShow		;
		//                                                  
		//lrDispencersCatchHeightSVShow						:=    VIS.lrDispencersCatchHeightSVShow				;  	// Pozycja chwytaka
		//lrDispencersLifterReadyPosition						:=    VIS.lrDispencersLifterReadyPositionShow		;
		
		iVirtualCycleCase									:=	 100;
	100:
		bRun												:=	TRUE;

		IF (tonChartRun.Q) AND fbDisp.eRunningState=5 THEN
			bRun											:=	FALSE;
			VIS.bDrawChart							:=	FALSE;
			iVirtualCycleCase								:=	0;
		END_IF
END_CASE

		VIS.aHorizontalChart[0][0]	:=VIS.nTimeMarkerDSPh5;		//najbardziej z tylu
		VIS.aHorizontalChart[1][0]	:=VIS.nTimeMarkerDSPh4;
		VIS.aHorizontalChart[2][0]	:=VIS.nTimeMarkerDSPh3;
		VIS.aHorizontalChart[3][0]	:=VIS.nTimeMarkerDSPh2;
		VIS.aHorizontalChart[4][0]	:=VIS.nTimeMarkerDSPh1;						//najbardziej z przodu
		



CASE VIS.udiDossagerNum OF

	0:	MEMCPY(ADR(VIS.aPoints),ADR(aPoints0),SIZEOF(VIS.aPoints));	//Show to wis
		VIS.nTimeMarkerDSPh1:=fbChart0.nTimeMarkerDSPh1;
		VIS.nTimeMarkerDSPh2:=fbChart0.nTimeMarkerDSPh2;
		VIS.nTimeMarkerDSPh3:=fbChart0.nTimeMarkerDSPh3;
		VIS.nTimeMarkerDSPh4:=fbChart0.nTimeMarkerDSPh4;
		VIS.nTimeMarkerDSPh5:=fbChart0.nTimeMarkerEnd+500;
		VIS.lrTorqMax		:=fbChart0.lrTorqMax;
		VIS.lrTorqMin		:=fbChart0.lrTorqMin;
	1:	MEMCPY(ADR(VIS.aPoints),ADR(aPoints1),SIZEOF(VIS.aPoints));	//Show to wis
		VIS.nTimeMarkerDSPh1:=fbChart1.nTimeMarkerDSPh1;
		VIS.nTimeMarkerDSPh2:=fbChart1.nTimeMarkerDSPh2;
		VIS.nTimeMarkerDSPh3:=fbChart1.nTimeMarkerDSPh3;
		VIS.nTimeMarkerDSPh4:=fbChart1.nTimeMarkerDSPh4;
		VIS.nTimeMarkerDSPh5:=fbChart1.nTimeMarkerEnd+500;
		VIS.lrTorqMax		:=fbChart1.lrTorqMax;		
		VIS.lrTorqMin		:=fbChart1.lrTorqMin;		
	2:	MEMCPY(ADR(VIS.aPoints),ADR(aPoints2),SIZEOF(VIS.aPoints));	//Show to wis
		VIS.nTimeMarkerDSPh1:=fbChart2.nTimeMarkerDSPh1;
		VIS.nTimeMarkerDSPh2:=fbChart2.nTimeMarkerDSPh2;
		VIS.nTimeMarkerDSPh3:=fbChart2.nTimeMarkerDSPh3;
		VIS.nTimeMarkerDSPh4:=fbChart2.nTimeMarkerDSPh4;
		VIS.nTimeMarkerDSPh5:=fbChart2.nTimeMarkerEnd+500;
		VIS.lrTorqMax		:=fbChart2.lrTorqMax;	
		VIS.lrTorqMin		:=fbChart2.lrTorqMin;		
	3:	MEMCPY(ADR(VIS.aPoints),ADR(aPoints3),SIZEOF(VIS.aPoints));	//Show to wis
        VIS.nTimeMarkerDSPh1:=fbChart3.nTimeMarkerDSPh1;
        VIS.nTimeMarkerDSPh2:=fbChart3.nTimeMarkerDSPh2;
		VIS.nTimeMarkerDSPh3:=fbChart3.nTimeMarkerDSPh3;
		VIS.nTimeMarkerDSPh4:=fbChart3.nTimeMarkerDSPh4;
		VIS.nTimeMarkerDSPh5:=fbChart3.nTimeMarkerEnd+500;
		VIS.lrTorqMax		:=fbChart3.lrTorqMax;
		VIS.lrTorqMin		:=fbChart3.lrTorqMin;		
END_CASE
END_ACTION

END_PROGRAM

// ---- POUs/FB/Charts/FB_ChartGenerator.TcPOU
FUNCTION_BLOCK FB_ChartGenerator
VAR_INPUT
	iCpuCycleTimeMs										:	INT:=3; //Czas TASK od CPU
	iTaskPerMesure										:	INT:=10;  //Ilość tasków na 1 punkt obliczenia
	bStrictMode											:	BOOL;
	bEnSim												:	BOOL;
END_VAR
VAR_OUTPUT
	nTimeMarkerEnd			:INT;
	nTimeMarkerDRPh1		:INT;
	nTimeMarkerDRPh2		:INT;	
	nTimeMarkerDRPh3		:INT;	
	nTimeMarkerDSPh1		:INT;	
	nTimeMarkerDSPh2		:INT;	
	nTimeMarkerDSPh3		:INT;
	nTimeMarkerDSPh4		:INT;
	lrTorqMin  : LREAL;
    lrTorqMax  : LREAL;
		
END_VAR
VAR
	actX												:	INT;
	h													:	INT;
	iMesureCounter										:	INT;
	rt_run												:	R_TRIG;
	rt_cd												:	R_TRIG;
	i													:	INT;
	k													:	INT;
	j													:	INT;
	bInit												:	BOOL;
	bFound   											: 	BOOL := FALSE;
	bFirstScan   										: 	BOOL := TRUE;
	rtSuckValve											:	R_TRIG;
	ftSuckValve											:	F_TRIG;		
	
	rtDoseValve											:	R_TRIG;
	ftDoseValve											:	F_TRIG;	
	
	rtPh1												:	R_TRIG;
	ftPh1                                               :	F_TRIG;
	
	rtPh2												:	R_TRIG;	
	ftPh2                                               :	F_TRIG;

	rtPh3												:	R_TRIG;
	ftPh3                                               :	F_TRIG;	
	rtGU	:R_trig;
	rt2Ph1												:	R_TRIG;
	ft2Ph1                                               :	F_TRIG;
	
	rt2Ph2												:	R_TRIG;	
	ft2Ph2                                               :	F_TRIG;

	rt2Ph3												:	R_TRIG;
	ft2Ph3                                               :	F_TRIG;
	
	ftPtR												:F_trig;
	
	actX2												:	INT;
	h2													:	INT;
	iMesureCounter2										:	INT;
	rt_run2												:	R_TRIG;
	rt_cd2												:	R_TRIG;
	i2													:	INT;
	k2													:	INT;
	j2													:	INT;
	bInit2												:	BOOL;
	aPointsBuf2											:	ARRAY [0..5,0..nPointarraySize-1] OF ST_Point;
	rt_copy2											:	R_TRIG;
	
	rtSuckValve2										:	R_TRIG;
	ftSuckValve2										:	F_TRIG;		
	
	rtDoseValve2										:	R_TRIG;
	ftDoseValve2										:	F_TRIG;	
	
END_VAR
VAR_IN_OUT
	aPointsBuf											:	ARRAY [0..11,0..nPointarraySize-1] OF ST_Point;
	fbDispencer											:	FB_ServoDispencerServoLifter;
	fbDispencer2										:	FB_ServoDispencerServoLifter;
	DispencerAxisRef       								: 	AXIS_REF; //Struktura sterowania NC dla serwa Dozownika
	DispencerAxisRef2       							: 	AXIS_REF; //Struktura sterowania NC dla serwa Dozownika
END_VAR
VAR CONSTANT 
	nAxisDispencer										:	INT := 0;
	nAxisLifter											:	INT := 1;	
	nSuckingValve										:	INT := 2;	
	nDosingValve										:	INT := 3;	
	nTimeMarks											:	INT := 4;	
	nAxisDispencer2										:	INT := 5;
	nAxisLifter2										:	INT := 6;	
	nSuckingValve2										:	INT := 7;	
	nDosingValve2										:	INT := 8;	
	nTimeMarks2											:	INT := 9;
	nAxisDispencerTorq									:	INT :=10;
	nAxisDispencerTorq2									:	INT :=11;
	
	nPointarraySize										:	INT := 600;

	nSuckingValveYoffset								:	INT := 50;	
	nDosingValveYoffset									:	INT := 10;	
	nValveOnYoffset										:	INT := 20;	
END_VAR

//Init
IF (NOT bInit) THEN
	
	FOR h:=0 TO 10 DO
		aPointsBuf[nTimeMarks,h * 3 + 0].y 							:= -10;	//Vertical line 1
		aPointsBuf[nTimeMarks,h * 3 + 1].y 							:= 500;
		aPointsBuf[nTimeMarks,h * 3 + 2].y 							:= -10;
		
		aPointsBuf[nTimeMarks2,h * 3 + 0].y 						:= -10;	//Vertical line 1
		aPointsBuf[nTimeMarks2,h * 3 + 1].y 						:= 500;
		aPointsBuf[nTimeMarks2,h * 3 + 2].y 						:= -10;
	END_FOR

	bInit												:= TRUE;
	
END_IF

rt_run		(CLK	:=	fbDispencer.bRun			);


//Hid all vertical lines and hide diagram
IF (rt_run.Q) THEN
	i:=0;
	
	FOR h:=0 TO 30 DO
		aPointsBuf[nTimeMarks,	h].x 					:= -1;
	END_FOR
	
	FOR k:=0 TO nPointarraySize-1 DO
		FOR j:=0 TO 3 DO
			aPointsBuf[j,	k].y 						:= 0;
		END_FOR
	END_FOR
	
END_IF

IF (fbDispencer.bRun AND i<nPointarraySize) THEN
	iMesureCounter										:=	iMesureCounter	+	1;
	IF (iMesureCounter>=iTaskPerMesure) THEN
		
		actX													:= i * iCpuCycleTimeMs * iTaskPerMesure ;
	
		rt_cd		(CLK	:=	fbDispencer.bCycleDone		);

		//Draw line CycleDone
		IF (rt_cd.Q) THEN
			aPointsBuf[nTimeMarks,	0].x 						:= actX;
			aPointsBuf[nTimeMarks,	1].x 						:= actX;
			aPointsBuf[nTimeMarks,	2].x 						:= actX;
		END_IF
	
		rtSuckValve(CLK:=fbDispencer.bSuckingValveActuator);
		IF (rtSuckValve.Q) THEN
			aPointsBuf[nTimeMarks,	3].x 						:= actX;
			aPointsBuf[nTimeMarks,	4].x 						:= actX;
			aPointsBuf[nTimeMarks,	5].x 						:= actX;
		END_IF
		
		ftSuckValve(CLK:=fbDispencer.bSuckingValveActuator);
		IF (ftSuckValve.Q) THEN
			aPointsBuf[nTimeMarks,	6].x 						:= actX;
			aPointsBuf[nTimeMarks,	7].x 						:= actX;
			aPointsBuf[nTimeMarks,	8].x 						:= actX;
		END_IF
		
		rtDoseValve(CLK:=fbDispencer.bDosingValveActuator);
		IF (rtDoseValve.Q) THEN
			aPointsBuf[nTimeMarks,	9].x 						:= actX;
			aPointsBuf[nTimeMarks,	10].x 						:= actX;
			aPointsBuf[nTimeMarks,	11].x 						:= actX;
		END_IF
		
		ftDoseValve(CLK:=fbDispencer.bDosingValveActuator);	
		IF (ftDoseValve.Q) THEN
			aPointsBuf[nTimeMarks,	12].x 						:= actX;
			aPointsBuf[nTimeMarks,	13].x 						:= actX;
			aPointsBuf[nTimeMarks,	14].x 						:= actX;
		END_IF
		
		rtPh1(Clk:=fbDispencer.eRunningState=7);
		ftPh2(Clk:=fbDispencer.eRunningState=8);
		IF (rtPh1.Q) THEN
			aPointsBuf[nTimeMarks,	15].x 						:= actX;
			aPointsBuf[nTimeMarks,	16].x 						:= actX;
			aPointsBuf[nTimeMarks,	17].x 						:= actX;
		END_IF
		IF (ftPh1.Q) THEN
			nTimeMarkerDRPh1:=actX;
		END_IF
		rtPh2(Clk:=fbDispencer.eRunningState=8);
		ftPh2(Clk:=fbDispencer.eRunningState=8);
		IF (rtPh2.Q) THEN
			aPointsBuf[nTimeMarks,	18].x 						:= actX;
			aPointsBuf[nTimeMarks,	19].x 						:= actX;
			aPointsBuf[nTimeMarks,	20].x 						:= actX;
		END_IF
		
		IF (ftPh2.Q) THEN
			nTimeMarkerDRPh2:= actX;
		END_IF
		
				
		rtPh3(Clk:=fbDispencer.eRunningState=9);
		ftPh3(Clk:=fbDispencer.eRunningState=9);
		IF (rtPh3.Q) THEN
			aPointsBuf[nTimeMarks,	21].x 						:= actX;
			aPointsBuf[nTimeMarks,	22].x 						:= actX;
			aPointsBuf[nTimeMarks,	23].x 						:= actX;
		END_IF

		IF (ftPh3.Q) THEN
			nTimeMarkerDRPh3:= actX;
		END_IF
	
		FOR j:=0 TO 3 DO
			aPointsBuf[j,i].x 									:= actX;
		END_FOR
			
		aPointsBuf[nAxisDispencer		,i].y			:=	LREAL_TO_INT(DispencerAxisRef.NcToPlc.ActPos);
		aPointsBuf[nAxisLifter			,i].y			:=	LREAL_TO_INT(fbDispencer.lrLifterActualPosition);
		aPointsBuf[nAxisDispencerTorq   ,i].y			:=	LREAL_TO_INT((DispencerAxisRef.NcToPlc.ActTorque/100)*9.8);
		aPointsBuf[nAxisDispencerTorq ,i].x := actX;
		
		IF (fbDispencer.bSuckingValveActuator) THEN
			aPointsBuf[nSuckingValve,	i].y 			:=	nSuckingValveYoffset + nValveOnYoffset;
		ELSE
			aPointsBuf[nSuckingValve,	i].y 			:= 	nSuckingValveYoffset;
		END_IF
	
		IF (fbDispencer.bDosingValveActuator) THEN
			aPointsBuf[nDosingValve,	i].y 			:= 	nDosingValveYoffset + nValveOnYoffset;
		ELSE
			aPointsBuf[nDosingValve,	i].y 			:= 	nDosingValveYoffset;
		END_IF
		
		FOR k:=i TO (nPointarraySize - 2) DO
			FOR j:=0 TO 3 DO
				aPointsBuf[j,k+1].y 					:=	aPointsBuf[j,k].y;
				aPointsBuf[j,k+1].x 					:=	aPointsBuf[j,k].x;
			END_FOR
			 aPointsBuf[nAxisDispencerTorq,k+1].y := aPointsBuf[nAxisDispencerTorq,k].y;
    		 aPointsBuf[nAxisDispencerTorq,k+1].x := aPointsBuf[nAxisDispencerTorq,k].x;
		END_FOR
	
		i												:=	i+1;
		iMesureCounter									:=	0;
	END_IF
	IF bFirstScan THEN
    	lrTorqMin := aPointsBuf[nAxisDispencerTorq, 0].y;
    	lrTorqMax := aPointsBuf[nAxisDispencerTorq, 0].y;
    	bFirstScan := FALSE;
	END_IF

	FOR h := 0 TO nPointarraySize - 1 DO
    // MIN
    IF aPointsBuf[nAxisDispencerTorq, h].y < lrTorqMin THEN
        lrTorqMin := aPointsBuf[nAxisDispencerTorq, h].y;
    END_IF

    // MAX
    IF aPointsBuf[nAxisDispencerTorq, h].y > lrTorqMax THEN
        lrTorqMax := aPointsBuf[nAxisDispencerTorq, h].y;
    END_IF
END_FOR

END_IF







rt_run2		(CLK	:=	fbDispencer2.bRun			);


//Hid all vertical lines and hide diagram
IF (rt_run2.Q  AND bEnSim) THEN
	i2:=0;
	
	FOR h2:=0 TO 30 DO
		aPointsBuf[nTimeMarks2,	h2].x 					:= -1;
	END_FOR
	
	FOR k2:=0 TO nPointarraySize-1 DO
		FOR j2:=5 TO 8 DO
			aPointsBuf[j2,	k2].y 						:= 0;
		END_FOR
	END_FOR
	
END_IF

IF (fbDispencer2.bRun AND i2<nPointarraySize) THEN
	iMesureCounter2										:=	iMesureCounter2	+	1;
	IF (iMesureCounter2>=iTaskPerMesure) THEN
		
		actX2													:= i2 * iCpuCycleTimeMs * iTaskPerMesure;
	
		rt_cd2		(CLK	:=	fbDispencer2.bCycleDone		);

		//Draw line CycleDone
		IF (rt_cd2.Q) THEN
			aPointsBuf[nTimeMarks2,	0].x 						:= actX2;
			aPointsBuf[nTimeMarks2,	1].x 						:= actX2;
			aPointsBuf[nTimeMarks2,	2].x 						:= actX2;
		END_IF
			nTimeMarkerEnd:=aPointsBuf[nTimeMarks2,	0].x;
			
		rtSuckValve2(CLK:=fbDispencer2.bSuckingValveActuator);
		IF (rtSuckValve2.Q) THEN
			aPointsBuf[nTimeMarks2,	3].x 						:= actX2;
			aPointsBuf[nTimeMarks2,	4].x 						:= actX2;
			aPointsBuf[nTimeMarks2,	5].x 						:= actX2;
		END_IF
		
		ftSuckValve2(CLK:=fbDispencer2.bSuckingValveActuator);
		IF (ftSuckValve2.Q) THEN
			aPointsBuf[nTimeMarks2,	6].x 						:= actX2;
			aPointsBuf[nTimeMarks2,	7].x 						:= actX2;
			aPointsBuf[nTimeMarks2,	8].x 						:= actX2;
		END_IF
		
		rtDoseValve2(CLK:=fbDispencer2.bDosingValveActuator);
		IF (rtDoseValve2.Q) THEN
			aPointsBuf[nTimeMarks2,	9].x 						:= actX2;
			aPointsBuf[nTimeMarks2,	10].x 						:= actX2;
			aPointsBuf[nTimeMarks2,	11].x 						:= actX2;
		END_IF
		
		ftDoseValve2(CLK:=fbDispencer2.bDosingValveActuator);	
		IF (ftDoseValve2.Q) THEN
			aPointsBuf[nTimeMarks2,	12].x 						:= actX2;
			aPointsBuf[nTimeMarks2,	13].x 						:= actX2;
			aPointsBuf[nTimeMarks2,	14].x 						:= actX2;
		END_IF
		ftPtR(Clk:=fbDispencer2.eRunningState=6);
		rt2Ph1(Clk:=fbDispencer2.eRunningState=7);
		ft2PH1(CLK:=fbDispencer2.eRunningState=7);
		IF (rt2Ph1.Q) THEN
			aPointsBuf[nTimeMarks2,	15].x 						:= actX2;
			aPointsBuf[nTimeMarks2,	16].x 						:= actX2;
			aPointsBuf[nTimeMarks2,	17].x 						:= actX2;
		END_IF		
			nTimeMarkerDSPh1:=aPointsBuf[nTimeMarks2,	16].x;
		IF VIS.lrDispencer1Phase1VolumeShow<1 THEN
			IF ftPtr.Q THEN
				nTimeMarkerDSPh2:=0;
			END_IF
		ELSE
			nTimeMarkerDSPh2:=aPointsBuf[nTimeMarks2,	19].x; //16
		END_IF
		

	
		rt2Ph2(Clk:=fbDispencer2.eRunningState=8);
		ft2PH2(CLK:=fbDispencer2.eRunningState=8);
		IF (rt2Ph2.Q) THEN
			aPointsBuf[nTimeMarks2,	18].x 						:= actX2;
			aPointsBuf[nTimeMarks2,	19].x 						:= actX2;
			aPointsBuf[nTimeMarks2,	20].x 						:= actX2;
		END_IF

		//	nTimeMarkerDSPh2:= aPointsBuf[nTimeMarks2,	19].x;

		rt2Ph3(Clk:=fbDispencer2.eRunningState=9);
		ft2PH3(CLK:=fbDispencer2.eRunningState=9);
		IF (rt2Ph3.Q) THEN
			aPointsBuf[nTimeMarks2,	21].x 						:= actX2;
			aPointsBuf[nTimeMarks2,	22].x 						:= actX2;
			aPointsBuf[nTimeMarks2,	23].x 						:= actX2;
		END_IF
		rtGU(CLK:=fbDispencer2.eRunningState=14);
		IF VIS.lrDispencer1Phase2VolumeShow<1 THEN
			IF rtGU.q THEN
				nTimeMarkerDSPh3:=actX2;
			END_IF
			nTimeMarkerDSPh4:=0;
		ELSE
			nTimeMarkerDSPh3:=aPointsBuf[nTimeMarks2,	22].x;
			IF rtgu.Q THEN
				nTimeMarkerDSPh4:=actX2;
			END_IF
		END_IF
		
		FOR j2:=5 TO 8 DO
			aPointsBuf[j2,i2].x 								:= actX2;
		END_FOR
			
		aPointsBuf[nAxisDispencer2		,i2].y			:=	LREAL_TO_INT(DispencerAxisRef2.NcToPlc.ActPos);
		aPointsBuf[nAxisLifter2			,i2].y			:=	LREAL_TO_INT(fbDispencer2.lrLifterActualPosition);
		aPointsBuf[nAxisDispencerTorq2			,i].y			:=	LREAL_TO_INT(DispencerAxisRef2.NcToPlc.ActTorque);
		
		IF (fbDispencer2.bSuckingValveActuator) THEN
			aPointsBuf[nSuckingValve2,	i2].y 			:=	nSuckingValveYoffset + nValveOnYoffset;
		ELSE
			aPointsBuf[nSuckingValve2,	i2].y 			:= 	nSuckingValveYoffset;
		END_IF
	
		IF (fbDispencer2.bDosingValveActuator) THEN
			aPointsBuf[nDosingValve2,	i2].y 			:= 	nDosingValveYoffset + nValveOnYoffset;
		ELSE
			aPointsBuf[nDosingValve2,	i2].y 			:= 	nDosingValveYoffset;
		END_IF
		aPointsBuf[nAxisDispencerTorq2, i2].y			:=0;
		aPointsBuf[nAxisDispencerTorq2, i2].x			:=actX2;
		FOR k2:=i2 TO (nPointarraySize - 2) DO
			FOR j2:=5 TO 8 DO
				aPointsBuf[j2,k2+1].y 					:=	aPointsBuf[j2,k2].y;
				aPointsBuf[j2,k2+1].x 					:=	aPointsBuf[j2,k2].x;
			END_FOR
			 aPointsBuf[nAxisDispencerTorq2,k2+1].y := aPointsBuf[nAxisDispencerTorq2,k2].y;
    		 aPointsBuf[nAxisDispencerTorq2,k2+1].x := aPointsBuf[nAxisDispencerTorq2,k2].x;
		END_FOR
	
		i2												:=	i2+1;
		iMesureCounter2									:=	0;
	END_IF
END_IF

END_FUNCTION_BLOCK

// ---- POUs/P00_PneumaticValves.TcPOU
(*
Nazwa:			P00_PneumaticValves
Opis:			Wyspa pneumatyczna
Wersja:			v1.0
Data:			2025-10-20
Autor:			DP
Urzadzenia:		Obsługa wyspy zaworowej
Konfiguracja:	
Info:
- kazdy zawór to 2 bity
#######################################################
#######################################################
*)



PROGRAM P00_PneumaticValves
VAR
	//ZMIENNE STERUJĄCE WYSPY ZAWOROWEJ
	QABPneumatic641ValveCoils 			AT %Q* 	: ARRAY[1..6] OF BYTE;
	QABPneumatic642ValveCoils 			AT %Q*	: ARRAY[1..5] OF BYTE;
	QABPneumatic643ValveCoils 			AT %Q*	: ARRAY[1..5] OF BYTE;
	QABPneumatic644ValveCoils 			AT %Q*	: ARRAY[1..5] OF BYTE;
	QABPneumatic645ValveCoils 			AT %Q*	: ARRAY[1..2] OF BYTE;
	QABPneumatic646ValveCoils 			AT %Q* 	: ARRAY[1..5] OF BYTE;
	QABPneumatic647ValveCoils 			AT %Q* 	: ARRAY[1..5] OF BYTE;
	QABPneumaticPI641ValveCoils 		AT %Q* 	: ARRAY[1..6] OF BYTE;

	QABPneumatic641PressureRegulator 	AT %Q* 	: ARRAY[1..2] OF BYTE;
	IABPneumatic641PressureRegulator 	AT %I* 	: ARRAY[1..2] OF BYTE;
	QABPneumatic645_1PressureRegulator 	AT %Q* 	: ARRAY[1..2] OF BYTE;
	IABPneumatic645_1PressureRegulator 	AT %I* 	: ARRAY[1..2] OF BYTE;
	QABPneumatic645_2PressureRegulator 	AT %Q* 	: ARRAY[1..2] OF BYTE;
	IABPneumatic645_2PressureRegulator 	AT %I* 	: ARRAY[1..2] OF BYTE;
	
	IABPneumatic641_N11AnalogInput1 	AT %I* 	: ARRAY[1..2] OF BYTE;
	IABPneumatic641_N11AnalogInput2 	AT %I* 	: ARRAY[1..2] OF BYTE;
	IABPneumatic641_N11AnalogInput3 	AT %I* 	: ARRAY[1..2] OF BYTE;
	IABPneumatic641_N11AnalogInput4 	AT %I* 	: ARRAY[1..2] OF BYTE;
	IABPneumatic645_N11AnalogInput1 	AT %I* 	: ARRAY[1..2] OF BYTE;
	IABPneumatic645_N11AnalogInput2 	AT %I* 	: ARRAY[1..2] OF BYTE;
	IABPneumatic645_N11AnalogInput3 	AT %I* 	: ARRAY[1..2] OF BYTE;
	IABPneumatic645_N11AnalogInput4 	AT %I* 	: ARRAY[1..2] OF BYTE;
	                                    
	IABPneumatic641_N12DigitalInput 	AT %I* 	: BYTE;	
	IABPneumatic642_N11DigitalInput 	AT %I* 	: BYTE;	
	IABPneumatic642_N12DigitalInput 	AT %I* 	: BYTE;	
	IABPneumatic642_N13DigitalInput 	AT %I* 	: BYTE;	
	IABPneumatic643_N11DigitalInput 	AT %I* 	: BYTE;	
	IABPneumatic643_N12DigitalInput 	AT %I* 	: BYTE;	
	IABPneumatic643_N13DigitalInput 	AT %I* 	: BYTE;
	IABPneumatic644_N11DigitalInput 	AT %I* 	: BYTE;	
	IABPneumatic644_N12DigitalInput 	AT %I* 	: BYTE;	
	IABPneumatic644_N13DigitalInput 	AT %I* 	: BYTE;
	IABPneumatic645_N12DigitalInput 	AT %I* 	: BYTE;
	IABPneumatic646_N11DigitalInput 	AT %I* 	: BYTE;
	IABPneumatic646_N12DigitalInput 	AT %I* 	: BYTE;
	IABPneumatic646_N13DigitalInput 	AT %I* 	: BYTE;
	IABPneumatic647_N11DigitalInput 	AT %I* 	: BYTE;
	IABPneumatic647_N12DigitalInput 	AT %I* 	: BYTE;
	IABPneumaticPI641_N11DigitalInput 	AT %I* 	: BYTE;
	IABPneumaticPI641_N12DigitalInput 	AT %I* 	: BYTE;
	IABPneumaticPI641_N13DigitalInput 	AT %I* 	: BYTE;
	                                  
	iIABPneumatic645_N11AnalogInput1	:INT;
	iIABPneumatic645_N11AnalogInput2    :INT;
	iIABPneumatic645_N11AnalogInput3    :INT;
	iIABPneumatic645_N11AnalogInput4    :INT;
	iIABPneumatic641_N11AnalogInput1    :INT;
	iIABPneumatic641_N11AnalogInput2    :INT;
	iIABPneumatic641_N11AnalogInput3    :INT;
	iIABPneumatic641_N11AnalogInput4    :INT;
	
	iIABPneumatic641PressureRegulator1				: INT;
	iIABPneumatic641PressureRegulator2				: INT;
	iIABPneumatic645_1PressureRegulator1			: INT;
	iIABPneumatic645_1PressureRegulator2			: INT;
	iIABPneumatic645_2PressureRegulator1			: INT;
	iIABPneumatic645_2PressureRegulator2			: INT;
	
	iQABPneumatic641PressureRegulator1				: INT;
	iQABPneumatic641PressureRegulator2				: INT;	
	iQABPneumatic645_1PressureRegulator1			: INT;
	iQABPneumatic645_1PressureRegulator2			: INT;
	iQABPneumatic645_2PressureRegulator1			: INT;
	iQABPneumatic645_2PressureRegulator2			: INT;	
	                                    
	(*Skalowanie czujników poziomu*)    
	fbiTank1LevelSensorValue 			: FB_4_20mA_TO_INT;
	fbiTank2LevelSensorValue 			: FB_4_20mA_TO_INT;	
	
	lrLidSealerPressureTemp						: LREAL;
	lrGripperScrewerCatchPressureTemp			: LREAL;
	lrGripperScrewerPressureTemp				: LREAL;
	lrDispencercatchPressureTemp				: LREAL;

	
END_VAR

//aVTEM();
//aVTEMSignals();
aAnalogueInput();
aDigitalInput();
aPressureRegulator();
aValveCoil();

ACTION aAnalogueInput:
(*
Nazwa:			aAnalogueInput
Opis:			Zawory pneumatyczne
Wersja:			v0.1
Data:			2024-10-28
Autor:			DP
Urzadzenia:		
Konfiguracja:	
Info:
- Czujnik pozycji Balluff, trzeba skonfigurować na 4-20mA, domyślnie jest na 0-10V
- Instrukcja konfiguracji czujnika: 2s, 1x, 1x (zniknie dioda), 2s (wyjście), 2s (wyjście)
*)

(*************************** 641N1.1 **************************************)
// Wyspa 1 - dozowanie
//AI1 4-20mA 
IABPneumatic641_N11AnalogInput1[1];
IABPneumatic641_N11AnalogInput1[2];
iIABPneumatic641_N11AnalogInput1	:= WORD_TO_INT(F_2Bytes_To_Word(byHigh:=IABPneumatic641_N11AnalogInput1[2],byLow:=IABPneumatic641_N11AnalogInput1[1]));
P02_Dispencers.IbDispencersCatch1SensorValue:=F_Scaling(rValue:=iIABPneumatic641_N11AnalogInput1, 
	rXmin:=		0,		//	0mA
	rXmax:=		32767,	//	23mA
	rYmin:= 	-70000, //	~10000 -> ~10mm (szyjka butelki) zamkniety (chwytak otwiera się na 49mm)
	rYmax:=		135000 );// ~60000 -> ~60mm otwarty
{warning 'dodać błąd czujnika poniżej 4mA i powyżej 20mA'}
IABPneumatic641_N11AnalogInput2[1]; 
IABPneumatic641_N11AnalogInput2[2];
iIABPneumatic641_N11AnalogInput2	:= WORD_TO_INT(F_2Bytes_To_Word(byHigh:=IABPneumatic641_N11AnalogInput2[2],byLow:=IABPneumatic641_N11AnalogInput2[1]));
P02_Dispencers.IbDispencersCatch2SensorValue:=F_Scaling(rValue:=iIABPneumatic641_N11AnalogInput2, 
	rXmin:=		0,		//	0mA
	rXmax:=		32767,	//	23mA
	rYmin:= 	-70000, //	~10000 -> ~10mm (szyjka butelki) zamkniety (chwytak otwiera się na 49mm)
	rYmax:=		135000 );// ~60000 -> ~60mm otwarty

IABPneumatic641_N11AnalogInput3[1]; 
IABPneumatic641_N11AnalogInput3[2]; 
iIABPneumatic641_N11AnalogInput3	:= WORD_TO_INT(F_2Bytes_To_Word(byHigh:=IABPneumatic641_N11AnalogInput3[2],byLow:=IABPneumatic641_N11AnalogInput3[1]));
P02_Dispencers.IbDispencersCatch3SensorValue:=F_Scaling(rValue:=iIABPneumatic641_N11AnalogInput3, 
	rXmin:=		0,		//	0mA
	rXmax:=		32767,	//	23mA
	rYmin:= 	-70000, //	~10000 -> ~10mm (szyjka butelki) zamkniety (chwytak otwiera się na 49mm)
	rYmax:=		135000 );// ~60000 -> ~60mm otwarty

IABPneumatic641_N11AnalogInput4[1]; 	
IABPneumatic641_N11AnalogInput4[2]; 
iIABPneumatic641_N11AnalogInput4	:= WORD_TO_INT(F_2Bytes_To_Word(byHigh:=IABPneumatic641_N11AnalogInput4[2],byLow:=IABPneumatic641_N11AnalogInput4[1]));
P02_Dispencers.IbDispencersCatch4SensorValue:=F_Scaling(rValue:=iIABPneumatic641_N11AnalogInput4, 
	rXmin:=		0,		//	0mA
	rXmax:=		32767,	//	23mA
	rYmin:= 	-70000, //	~10000 -> ~10mm (szyjka butelki) zamkniety (chwytak otwiera się na 49mm)
	rYmax:=		135000 );// ~60000 -> ~60mm otwarty

(*********************Koniec 641N1.1 **************************************)


(*************************** 645N1.1 **************************************)
// Wyspa 5 - zakręcarki i czujnik poziomu
//AI1 4-20mA 
IABPneumatic645_N11AnalogInput1[1];
IABPneumatic645_N11AnalogInput1[2];
iIABPneumatic645_N11AnalogInput1	:= WORD_TO_INT(F_2Bytes_To_Word(byHigh:=IABPneumatic645_N11AnalogInput1[2],byLow:=IABPneumatic645_N11AnalogInput1[1]));
P10_GripperScrewer.IlrGripperScrewer1HeightCV	:=	-0.0023*(iIABPneumatic645_N11AnalogInput1)+52.006 + 2.6788;

IABPneumatic645_N11AnalogInput2[1]; 
IABPneumatic645_N11AnalogInput2[2]; 
iIABPneumatic645_N11AnalogInput2	:= WORD_TO_INT(F_2Bytes_To_Word(byHigh:=IABPneumatic645_N11AnalogInput2[2],byLow:=IABPneumatic645_N11AnalogInput2[1]));
P10_GripperScrewer.IlrGripperScrewer2HeightCV	:=	-0.0023*(iIABPneumatic645_N11AnalogInput2)+52.006 + 2.252;

IABPneumatic645_N11AnalogInput3[1];
IABPneumatic645_N11AnalogInput3[2];
iIABPneumatic645_N11AnalogInput3	:= WORD_TO_INT(F_2Bytes_To_Word(byHigh:=IABPneumatic645_N11AnalogInput3[2],byLow:=IABPneumatic645_N11AnalogInput3[1]));
//iTank1Sensor1Value;//Czujnik poziomu 1
fbiTank1LevelSensorValue(
	iIN:= 	iIABPneumatic645_N11AnalogInput3, 
	rXmin:= 5190,//5513.0, 	// 4mA
	rXmax:= 27307.0, 	// 20mA
	rYmin:= 10.0, 		// 10mm na czujniku to 4mA
	rYmax:= 325.0,		// 325mm na czujniku to 20mA
	bError=>, 			// Bląd <4mA i >20mA
	iOUT=>	VIS.iTank1LevelSensorValue );
fbiTank1LevelSensorValue.bError;

IABPneumatic645_N11AnalogInput4[1];
IABPneumatic645_N11AnalogInput4[2];
iIABPneumatic645_N11AnalogInput4	:= WORD_TO_INT(F_2Bytes_To_Word(byHigh:=IABPneumatic645_N11AnalogInput4[2],byLow:=IABPneumatic645_N11AnalogInput4[1]));
//iTank2Sensor2Value;//Czujnik poziomu 2
fbiTank2LevelSensorValue(
	iIN:= 	iIABPneumatic645_N11AnalogInput4, 
	rXmin:= 5190,//5513.0, 	// 4mA
	rXmax:= 27307.0, 	// 20mA
	rYmin:= 10.0, 		// 10mm na czujniku to 4mA
	rYmax:= 325.0,		// 325mm na czujniku to 20mA
	bError=>, 			// Bląd <4mA i >20mA
	iOUT=>	VIS.iTank2LevelSensorValue );
fbiTank2LevelSensorValue.bError;
END_ACTION

ACTION aDigitalInput:
(*
Nazwa:			aDigitalInput
Opis:			Wejścia podłączone do wyspy pneumatycznej
Wersja:			v0.1
Data:			2024-10-28
Autor:			DP
Urzadzenia:		
Konfiguracja:	
Info:
*)
(* Stare z UBL50 Ziaja
(*************************** A3 **************************************)
// Wyspa 7 - podajnik opakowań
MAIN.IbLidSealerAfterSensor:=IABPneumaticA3DigitalInput[1].7;   //brak czujnika, póki co nie dokładamy
MAIN.IbBlowBeforeGripperScrewerSensor  :=	IABPneumaticA3DigitalInput[2].1;	  //czujnik pomiędzy UL a UF -> (opcja) być moze do usunięcia
MAIN.IbCapSorterFirstFormCheckFormSensor := IABPneumaticA3DigitalInput[2].2;	
MAIN.IbCapSorterAfterFormSensor2 :=	IABPneumaticA3DigitalInput[2].3;	//Czujnik drag sortera nakretek	

*)

(*************************** 641N1.2 **************************************)
P02_Dispencers.IbDispencer1DropCatcherBackSensor		:=	IABPneumatic641_N12DigitalInput.0;
P02_Dispencers.IbDispencer2DropCatcherBackSensor		:=	IABPneumatic641_N12DigitalInput.1;
P02_Dispencers.IbDispencer3DropCatcherBackSensor		:=	IABPneumatic641_N12DigitalInput.2;
P02_Dispencers.IbDispencer4DropCatcherBackSensor		:=	IABPneumatic641_N12DigitalInput.3;
P01_BottleFeeder.IbBottleFeederNotInsertedSensor		:=	IABPneumatic641_N12DigitalInput.4;
GVL_IO.IbPressureInSystemSensor							:=  IABPneumatic641_N12DigitalInput.5; //ciśnienie robocze ok za zaworem bezpieczęństwa? 
P02_Dispencers.IbDispencer12NoColisionWhenDosingSensor	:=	IABPneumatic641_N12DigitalInput.6; //rezerwa
P02_Dispencers.IbDispencer34NoColisionWhenDosingSensor	:=	IABPneumatic641_N12DigitalInput.7; //rezerwa

(*************************** 642N1.1 **************************************)
P16_LabelMachine.IbLabelMachineFullSensor			:=	IABPneumatic642_N11DigitalInput.0;
P14_BadBottleConyevor.IbBadBottleConveyorFullSensor	:=	IABPneumatic642_N11DigitalInput.1;
MAIN.IbBottleInFormCheckBottleSensor				:=	IABPneumatic642_N11DigitalInput.2;
P13_BottleTransfer.IbBottleCheckAfterBottleTransferSensor	:=	IABPneumatic642_N11DigitalInput.3;
MAIN.IbFormCheckFormSensor							:=	IABPneumatic642_N11DigitalInput.4;
MAIN.IbFourthFormCheckFormSensor					:=	IABPneumatic642_N11DigitalInput.5;
MAIN.IbSecondFormCheckFormSensor			:=	IABPneumatic642_N11DigitalInput.6;	
P02_Dispencers.IbDispencerAfterCheckFormSensor		:=	IABPneumatic642_N11DigitalInput.7;

(*************************** 642N1.2 **************************************)
P13_BottleTransfer.IbFirstFormCheckFormSensor		:=	IABPneumatic642_N12DigitalInput.0;
P13_BottleTransfer.IbSecondFormCheckFormSensor	:=	IABPneumatic642_N12DigitalInput.1;
P13_BottleTransfer.IbBottleTransferFormAfterSensor	:=	IABPneumatic642_N12DigitalInput.2;
P13_BottleTransfer.IbBottleTransferFormAfterSensor2	:=	IABPneumatic642_N12DigitalInput.3;	//czujnik nr 2 kolejki za robotem ?
P01_TwoPhasesBarriers.IbBarrierBetweenDispencerOpenedSensor	:=	IABPneumatic642_N12DigitalInput.4;
P01_TwoPhasesBarriers.IbBarrierBetweenDispencerClosedSensor	:=	IABPneumatic642_N12DigitalInput.5;
P01_TwoPhasesBarriers.IbBarrierBetweenWeightOpenedSensor	:=	IABPneumatic642_N12DigitalInput.6;
P01_TwoPhasesBarriers.IbBarrierBetweenWeightClosedSensor	:=	IABPneumatic642_N12DigitalInput.7;

(*************************** 642N1.3 **************************************)
P02_Dispencers.IbDispencersDragLeftDragUpSensor			:=	IABPneumatic642_N13DigitalInput.0;
P02_Dispencers.IbDispencersDragLeftDragDownSensor		:=	IABPneumatic642_N13DigitalInput.1;
P02_Dispencers.IbDispencersDragLeftDragHomingSensor		:=	IABPneumatic642_N13DigitalInput.2;
P02_Dispencers.IbDispencersDragRightDragUpSensor		:=	IABPneumatic642_N13DigitalInput.3;
P02_Dispencers.IbDispencersDragRightDragDownSensor		:=	IABPneumatic642_N13DigitalInput.4;
P02_Dispencers.IbDispencersDragRightDragHomingSensor	:=	IABPneumatic642_N13DigitalInput.5;
P02_Dispencers.IbDispencersDragLeftLeadBefore1UpSensor	:=	IABPneumatic642_N13DigitalInput.6;
P02_Dispencers.IbDispencersDragRightLeadBefore1UpSensor	:=	IABPneumatic642_N13DigitalInput.7;

(*************************** 643N1.1 **************************************)
MAIN.IbTwoPhasesFormSensorBetweenDispencers		:=	IABPneumatic643_N11DigitalInput.0;
P01_Gates.IbGateBeforeWeights14Sensor			:=	IABPneumatic643_N11DigitalInput.1;							//obecność formatki przy rfid za 1 faza dozowniki
P01_Gates.IbGateBeforeWeights56Sensor			:=	IABPneumatic643_N11DigitalInput.2;							//obecność formatki przy rfid za 2 faza dozowniki
P05_Weight.IbWeight1FormSensor					:=	IABPneumatic643_N11DigitalInput.3;
P05_Weight.IbWeight2FormSensor					:=	IABPneumatic643_N11DigitalInput.4;
P05_Weight.IbWeight3FormSensor					:=	IABPneumatic643_N11DigitalInput.5;
P05_Weight.IbWeight4FormSensor					:=	IABPneumatic643_N11DigitalInput.6;
P06_LidFeeder.IbLidFeederFirstFormSensorBeforeDrag	:=	IABPneumatic643_N11DigitalInput.7;								//obecność 1 formatki przed podawaniem platynek
;
(*************************** 643N1.2 **************************************)
MAIN.IbLidFeederThirdFormSensor	:=	IABPneumatic643_N12DigitalInput.0;									//obecność 2 formatki przed podawaniem platynek
MAIN.IbLidFeederAfterSensor	:=	IABPneumatic643_N12DigitalInput.1;									//obecność formatki przy rfid przed przygrzewaniem platynek
P11_CapCorrectCheck.IbCapCorrectCheckAfterScrewerFormSensor	:=	IABPneumatic643_N12DigitalInput.2;		//kolejka formatek za zakręcarkami
P11_CapCorrectCheck.IbCapCorrectCheckFormSensor	:=	IABPneumatic643_N12DigitalInput.3;									//obecność formatki przy rfid kontrola zamknięcia	
P11_CapCorrectCheck.IbCapCorrectCheckBottleSensor	:=	IABPneumatic643_N12DigitalInput.4;		
P05_Weight.IbWeight6FormSensor :=	IABPneumatic643_N12DigitalInput.5;									
P05_Weight.IbWeight5FormSensor :=	IABPneumatic643_N12DigitalInput.6;									
IABPneumatic643_N12DigitalInput.7;										//rezerwa

(*************************** 643N1.3 **************************************)
IABPneumatic643_N13DigitalInput.0;	//szlaban przed wagami 1-4
P01_TwoPhasesBarriers.IbGateBeforeWeights56		:=	IABPneumatic643_N13DigitalInput.1;
P02_Dispencers.IbDispencersDragLeftLeadAfter1UpSensor		:=	IABPneumatic643_N13DigitalInput.2;
P02_Dispencers.IbDispencersDragRightLeadAfter1UpSensor		:=	IABPneumatic643_N13DigitalInput.3;
MAIN.IbLidSealerFirstFormSensor		:=	IABPneumatic643_N13DigitalInput.4;		// Czujnik obecności 1-ej formatki przygrzewacze platynek
MAIN.IbLidSealerSecondFormSensor	:=	IABPneumatic643_N13DigitalInput.5;	// Czujnik obecności 2-ej formatki przygrzewacze platynek 
IABPneumatic643_N13DigitalInput.6;	//rezerwa
IABPneumatic643_N13DigitalInput.7;	//rezerwa

(*************************** 644N1.1 **************************************)
MAIN.IbLidSealerAfterSensor	:=	IABPneumatic644_N11DigitalInput.0;									//czujnik formatki za przygrzewaczami
P10_GripperScrewer.IbGripperScrewersSixthFormCheckFormSensor		:=	IABPneumatic644_N11DigitalInput.1;	
P09_CapPuttedCheck.IbCapPuttedCheckFormSensor	:=	IABPneumatic644_N11DigitalInput.2;									//obecność formatki przy rfid przed zakręcarkami
P10_GripperScrewer.IbGripperScrewersBeforeThirdFormCheckFormSensor 	:=	IABPneumatic644_N11DigitalInput.3;
P10_GripperScrewer.IbGripperScrewersThirdFormCheckFormSensor		:=	IABPneumatic644_N11DigitalInput.4;
P11_CapCorrectCheck.IbCapCorrectCheckDialAfterScrewerFormSensor		:=	IABPneumatic644_N11DigitalInput.5;
P01_Gates.IbLidFeederBarrierOnSensor								:=	IABPneumatic644_N11DigitalInput.6;	//banda opuszczona pomiędzy podawaniem a przygrzewaniem platynek
P01_Gates.IbLidFeederBarrierOffSensor								:=	IABPneumatic644_N11DigitalInput.7;	//banda podniesiona pomiędzy podawaniem a przygrzewaniem platynek

(*************************** 644N1.2 **************************************)
//Platynki
(*P06_LidFeeder.IbLidFeederFormPositioning1HideSensor	:=	IABPneumatic644_N12DigitalInput.0;	//pozycjonowanie formatki pod podajnikiem platynek wsynięte
P06_LidFeeder.IbLidFeederFormPositioning2HideSensor	:=	IABPneumatic644_N12DigitalInput.1;	//pozycjonowanie formatki pod podajnikiem platynek wysunięte
P06_LidFeeder.IbLidFeederDragLeadBefore1UpSensor	:=	NOT IABPneumatic644_N12DigitalInput.2;
P06_LidFeeder.IbLidFeederDragUpSensor				:=	IABPneumatic644_N12DigitalInput.3;
P06_LidFeeder.IbLidFeederDragDownSensor				:=	IABPneumatic644_N12DigitalInput.4;
P06_LidFeeder.IbLidFeederDragHomingSensor			:=	IABPneumatic644_N12DigitalInput.5;
P06_LidSealer.IbLidSealerDragLeadBefore1UpSensor	:=	NOT IABPneumatic644_N12DigitalInput.6;
P06_LidSealer.IbLidSealerDragUpSensor				:=	IABPneumatic644_N12DigitalInput.7;*)
//Podajnik knotów
P06_WickFeeder.IbFormPositioningHide1				:=	IABPneumatic644_N12DigitalInput.0;	//pozycjonowanie formatki pod podajnikiem platynek wsynięte
P06_WickFeeder.IbFormPositioningHide2				:=	IABPneumatic644_N12DigitalInput.1;	//pozycjonowanie formatki pod podajnikiem platynek wysunięte
P06_WickFeeder.IbWickFeederDragLeadBefore1UpSensor	:=	IABPneumatic644_N12DigitalInput.2;
P06_WickFeeder.IbWickFeederDragUpSensor				:=	IABPneumatic644_N12DigitalInput.3;
P06_WickFeeder.IbWickFeederDragDownSensor			:=	IABPneumatic644_N12DigitalInput.4;
P06_WickFeeder.IbWickFeederDragHomingSensor			:=	IABPneumatic644_N12DigitalInput.5;
P06_LidSealer.IbLidSealerDragLeadBefore1UpSensor	:=	IABPneumatic644_N12DigitalInput.6;
P06_LidSealer.IbLidSealerDragUpSensor				:=	IABPneumatic644_N12DigitalInput.7;
(*************************** 644N1.3 **************************************)
P06_LidSealer.IbLidSealerDragDownSensor						:=	IABPneumatic644_N13DigitalInput.0;
P06_LidSealer.IbLidSealerDragHomingSensor					:=	IABPneumatic644_N13DigitalInput.1;
P10_GripperScrewer.IbGripperScrewersDragLeadBefore1UpSensor	:=	IABPneumatic644_N13DigitalInput.2;
P10_GripperScrewer.IbGripperScrewersDragLeadBefore2UpSensor	:=	IABPneumatic644_N13DigitalInput.3;
P10_GripperScrewer.IbGripperScrewersDragUpSensor			:=	IABPneumatic644_N13DigitalInput.4;
P10_GripperScrewer.IbGripperScrewersDragDownSensor			:=	IABPneumatic644_N13DigitalInput.5;
P10_GripperScrewer.IbGripperScrewersDragHomingSensor		:=	IABPneumatic644_N13DigitalInput.6;
IABPneumatic644_N13DigitalInput.7;	//rezerwa

(*************************** 645N1.2 **************************************)
P09_CapPuttedCheck.IbCapPuttedCheckSensor					:=	IABPneumatic645_N12DigitalInput.0;
P11_CapCorrectCheck.IbCapCorrectCheckCapOKSensor			:=	IABPneumatic645_N12DigitalInput.1;
P11_CapCorrectCheck.IbCapCorrectCheckCapNotScrewedSensor	:=	IABPneumatic645_N12DigitalInput.2;
IABPneumatic645_N12DigitalInput.3;	//chwytak zakręcarki otwarty				//brak fizycznie !!
IABPneumatic645_N12DigitalInput.4;	//chwytak zakręcarki zamknięty              //brak fizycznie !!
IABPneumatic645_N12DigitalInput.5;	//rezerwa
IABPneumatic645_N12DigitalInput.6;	//rezerwa
IABPneumatic645_N12DigitalInput.7;	//rezerwa

(*************************** 646N1.1 **************************************)
//Platynki
(*P06_LidFeeder.IbLidFeederUpSensor2		:=	IABPneumatic646_N11DigitalInput.0;	//głowica wieczek 1 u góry
P06_LidFeeder.IbLidFeederDownSensor2	:=	IABPneumatic646_N11DigitalInput.1;  //głowica wieczek 1 w dole
P06_LidFeeder.IbLidFeederUpSensor1		:=	IABPneumatic646_N11DigitalInput.2;  //głowica wieczek 2 u góry
P06_LidFeeder.IbLidFeederDownSensor1	:=	IABPneumatic646_N11DigitalInput.3;  //głowica wieczek 2 w dole
P06_LidFeeder.IbLidFeederLowLevelSensor2 :=	NOT IABPneumatic646_N11DigitalInput.4;  //obecność wieczek zbiornik 1
P06_LidFeeder.IbLidFeederLowLevelSensor1 :=	NOT IABPneumatic646_N11DigitalInput.5;  //obecność wieczek zbiornik 2
P06_LidFeeder.IbLidFeeder2SuckerSensor			:= IABPneumatic646_N11DigitalInput.6;  //rezerwa    //podciśnienie podsysania wieczka OK
P06_LidFeeder.IbLidFeederSuckerSensor	:=	IABPneumatic646_N11DigitalInput.7;  //rezerwa	//podciśnienie podsysania wieczka OK

IABPneumatic646_N12DigitalInput.0;	//rezerwa
IABPneumatic646_N12DigitalInput.1;  //rezerwa
IABPneumatic646_N12DigitalInput.2;  //rezerwa
IABPneumatic646_N12DigitalInput.3;  //rezerwa
IABPneumatic646_N12DigitalInput.4;  //rezerwa
IABPneumatic646_N12DigitalInput.5;  //rezerwa
IABPneumatic646_N12DigitalInput.6;  //rezerwa
IABPneumatic646_N12DigitalInput.7;  //rezerwa*)
//Knoty
P06_WickFeeder.IbQueFullSensor															:=	IABPneumatic646_N11DigitalInput.0;	
P06_WickFeeder.IbWheelSensor															:=	IABPneumatic646_N11DigitalInput.1; 
P06_WickFeeder.IbWheelLevelSensor														:=	IABPneumatic646_N11DigitalInput.2;  
P06_WickFeeder.IbWickAtPipe																:=	IABPneumatic646_N11DigitalInput.3;  
P06_WickFeeder.IbSeparatorPos1															:=	IABPneumatic646_N11DigitalInput.4;  
P06_WickFeeder.IbSeparatorPos2															:=		IABPneumatic646_N11DigitalInput.5;  
P06_WickFeeder.IbSleve1SeparatorOut														:= IABPneumatic646_N11DigitalInput.6; 
P06_WickFeeder.IbQueFullAtSleve1														:=	IABPneumatic646_N11DigitalInput.7; 

P06_WickFeeder.IbSleve2SeparatorOut														:=	IABPneumatic646_N12DigitalInput.0;	
P06_WickFeeder.IbQueFullAtSleve2														:=	IABPneumatic646_N12DigitalInput.1;  
P06_WickFeeder.IbWickAtSleve1															:=	IABPneumatic646_N12DigitalInput.2;  
P06_WickFeeder.IbWickAtSleve2															:=	IABPneumatic646_N12DigitalInput.3;  
P06_WickFeeder.IbHammer1Down															:=	IABPneumatic646_N12DigitalInput.4;  
P06_WickFeeder.IbHammer1Up																:=	IABPneumatic646_N12DigitalInput.5;  
P06_WickFeeder.IbHammer2Down															:=	IABPneumatic646_N12DigitalInput.6;  
P06_WickFeeder.IbHammer2Up																:=	IABPneumatic646_N12DigitalInput.7;  

P06_WickFeeder.IbQueFullAfterWheelSensor 												:=	IABPneumatic646_N13DigitalInput.0;	
IABPneumatic646_N13DigitalInput.1;  
IABPneumatic646_N13DigitalInput.2;  
IABPneumatic646_N13DigitalInput.3;  
IABPneumatic646_N13DigitalInput.4;  
IABPneumatic646_N13DigitalInput.5;  
IABPneumatic646_N13DigitalInput.6;  
IABPneumatic646_N13DigitalInput.7;  


(*************************** A3 **************************************)
// Wyspa 7 - podajnik opakowań
//DI1
P08_CapSorter.IbCapSorterDragUpSensor:=  IABPneumatic647_N11DigitalInput.0;	// widły pod podajnikiem zamknięć wysunięte
P08_CapSorter.IbCapSorterDragDownSensor:=  IABPneumatic647_N11DigitalInput.1;	 //widły pod podajnikiem zamknięć schowane
P08_CapSorter.IbCapSorterDragHomingSensor:= IABPneumatic647_N11DigitalInput.2;	//prowadzenie formatek przed podajnikiem zamknięć lewe podniesione
P08_CapSorter.IbCapSorterDragLeadBefore1UpSensor:=  IABPneumatic647_N11DigitalInput.3;	//prowadzenie formatek przed podajnikiem zamknięć lewe podniesione
P08_CapSorter.IbCapSorterDragLeadBefore2UpSensor:=  IABPneumatic647_N11DigitalInput.4;	//prowadzenie formatek przed podajnikiem zamknięć prawe podniesione
P08_CapSorter.IbCapSorterDragLeadAfter1UpSensor:=IABPneumatic647_N11DigitalInput.5;	//czujnik wjazdu przed podajnikiem zamknięć 
P08_CapSorter.IbCapSorterDragLeadAfter2UpSensor:=IABPneumatic647_N11DigitalInput.6;	// czujnik  4 formatki za podajnikiem zamknięć -> czujnik na ukos
;IABPneumatic647_N11DigitalInput.7;   //brak czujnika, póki co nie dokładamy
//DI2
MAIN.IbCapSorterFirstFormCheckFormSensor := IABPneumatic647_N12DigitalInput.0;	   //ostatnia formatka przed przeciąganiem
MAIN.IbCapSorterAfterFormSensor2  :=	IABPneumatic647_N12DigitalInput.1;	  //czujnik pomiędzy UL a UF -> (opcja) być moze do usunięcia
MAIN.IbCapSorterBeforeFourthFormCheckFormSensor := IABPneumatic647_N12DigitalInput.2;	
MAIN.IbCapSorterFourthFormCheckFormSensor :=	IABPneumatic647_N12DigitalInput.3;	//Czujnik drag sortera nakretek
MAIN.IbBlowBeforeGripperScrewerSensor := IABPneumatic647_N12DigitalInput.4;	
MAIN.IbCapSorterAfterFormSensor := IABPneumatic647_N12DigitalInput.5;		
IABPneumatic647_N12DigitalInput.6;		
IABPneumatic647_N12DigitalInput.7;		

(*********************Koniec A3 **************************************)

(*************************** 641**************************************)
// Wyspa 6 - podajnik opakowań
P01_pucksInserter.IbPucksInserterLevelSensor				:= IABPneumaticPI641_N11DigitalInput.0;	
P01_pucksInserter.IbPucksInserterWheelEntrySensor			:= IABPneumaticPI641_N11DigitalInput.1;	
P01_pucksInserter.IbPucksInserterWheelExitSensor			:= IABPneumaticPI641_N11DigitalInput.2;	
P01_pucksInserter.IbPucksInserterFormGateBeforeSensor		:= IABPneumaticPI641_N11DigitalInput.3;	
P01_pucksInserter.IbPucksInserterFormGateAfterSensor		:= IABPneumaticPI641_N11DigitalInput.4;	//czujnik kolejki Stołu podającego
P01_pucksInserter.IbPucksInserterHammerUpSensor				:= IABPneumaticPI641_N11DigitalInput.5;		
P01_pucksInserter.IbPucksInserterHammerDownSensor			:= IABPneumaticPI641_N11DigitalInput.6;		
P01_pucksInserter.IbPucksInserterTrayOffSensor				:= IABPneumaticPI641_N11DigitalInput.7;	
//DI2
P01_pucksInserter.IbPucksInserterTrayOnSensor				:= IABPneumaticPI641_N12DigitalInput.0;	
P01_pucksInserter.IbPucksInserterFormPositioningOffSensor	:= IABPneumaticPI641_N12DigitalInput.1;	
P01_pucksInserter.IbPucksInserterFormPositioningOnSensor	:= IABPneumaticPI641_N12DigitalInput.2;	
P01_pucksInserter.IbPucksInserterGate1OffSensor				:= IABPneumaticPI641_N12DigitalInput.3;	
P01_pucksInserter.IbPucksInserterGate1OnSensor				:= IABPneumaticPI641_N12DigitalInput.4;	
P01_pucksInserter.IbPucksInserterGate2OffSensor				:= IABPneumaticPI641_N12DigitalInput.5;
P01_pucksInserter.IbPucksInserterGate2OnSensor				:= IABPneumaticPI641_N12DigitalInput.6;		
P01_pucksInserter.IbPucksInserterHomingSensor				:= IABPneumaticPI641_N12DigitalInput.7;	

 P01_pucksInserter.IbPucksInserterPushTablesSensor			:= IABPneumaticPI641_N13DigitalInput.0;	
 IABPneumaticPI641_N13DigitalInput.1;	
 IABPneumaticPI641_N13DigitalInput.2;	
 IABPneumaticPI641_N13DigitalInput.3;	
 IABPneumaticPI641_N13DigitalInput.4;	
 IABPneumaticPI641_N13DigitalInput.5;
 IABPneumaticPI641_N13DigitalInput.6;	
 IABPneumaticPI641_N13DigitalInput.7;	



(*********************Koniec 641 **************************************)
END_ACTION

ACTION aPressureRegulator:
(*
Nazwa:			aPressureRegulator
Opis:			Zawory pneumatyczne
Wersja:			v1.0
Data:			2025-10-20
Autor:			DP
Urzadzenia:		
Konfiguracja:	
Info:
*)
IF VIS.lrDispencerCatchPressureShow <3.5 THEN
	VIS.lrDispencerCatchPressureShow  :=5;
END_IF
IF VIS.lrDispencerCatchPressureShow >12 THEN
	VIS.lrDispencerCatchPressureShow  :=12;
END_IF

lrDispencercatchPressureTemp := ((lrDispencerCatchPressure*10)/14.8)*1000;
lrGripperScrewerCatchPressureTemp := ((lrGripperScrewerCatchPressure*10)/26.2)*1000;
lrGripperScrewerPressureTemp := ((lrGripperScrewerPressure*10)/14.8)*1000;

iQABPneumatic641PressureRegulator1 := LREAL_TO_INT(lrDispencercatchPressureTemp);
iQABPneumatic645_1PressureRegulator1 := LREAL_TO_INT(lrGripperScrewerCatchPressureTemp);
iQABPneumatic645_2PressureRegulator2 := LREAL_TO_INT(lrGripperScrewerPressureTemp);
	
(*************************** 641 **************************************)
// Wyspa 1 - dozowanie
QABPneumatic641PressureRegulator[1].0		:= iQABPneumatic641PressureRegulator1.0; 
QABPneumatic641PressureRegulator[1].1		:= iQABPneumatic641PressureRegulator1.1;                 
QABPneumatic641PressureRegulator[1].2		:= iQABPneumatic641PressureRegulator1.2;
QABPneumatic641PressureRegulator[1].3		:= iQABPneumatic641PressureRegulator1.3;
QABPneumatic641PressureRegulator[1].4		:= iQABPneumatic641PressureRegulator1.4;
QABPneumatic641PressureRegulator[1].5		:= iQABPneumatic641PressureRegulator1.5;
QABPneumatic641PressureRegulator[1].6		:= iQABPneumatic641PressureRegulator1.6;
QABPneumatic641PressureRegulator[1].7		:= iQABPneumatic641PressureRegulator1.7;
QABPneumatic641PressureRegulator[2].0		:= iQABPneumatic641PressureRegulator1.8; 
QABPneumatic641PressureRegulator[2].1		:= iQABPneumatic641PressureRegulator1.9;                 
QABPneumatic641PressureRegulator[2].2		:= iQABPneumatic641PressureRegulator1.10;
QABPneumatic641PressureRegulator[2].3		:= iQABPneumatic641PressureRegulator1.11;
QABPneumatic641PressureRegulator[2].4		:= iQABPneumatic641PressureRegulator1.12;
QABPneumatic641PressureRegulator[2].5		:= iQABPneumatic641PressureRegulator1.13;
QABPneumatic641PressureRegulator[2].6		:= iQABPneumatic641PressureRegulator1.14;
QABPneumatic641PressureRegulator[2].7		:= iQABPneumatic641PressureRegulator1.15;

IABPneumatic641PressureRegulator[1];
IABPneumatic641PressureRegulator[2];
iIABPneumatic641PressureRegulator1	:= WORD_TO_INT(F_2Bytes_To_Word(byHigh:=IABPneumatic641PressureRegulator[2],byLow:=IABPneumatic641PressureRegulator[1]));

(*********************Koniec 641 **************************************)

(*************************** 645 **************************************)
// Wyspa 5 - zakręcarki

//PR1
QABPneumatic645_1PressureRegulator[1];
QABPneumatic645_1PressureRegulator[2];
//Zawór proporcjonalny chwytaki pod zakręcarkami szczękowymi
QABPneumatic645_1PressureRegulator[1].0		:= iQABPneumatic645_1PressureRegulator1.0; 
QABPneumatic645_1PressureRegulator[1].1		:= iQABPneumatic645_1PressureRegulator1.1;                 
QABPneumatic645_1PressureRegulator[1].2		:= iQABPneumatic645_1PressureRegulator1.2;
QABPneumatic645_1PressureRegulator[1].3		:= iQABPneumatic645_1PressureRegulator1.3;
QABPneumatic645_1PressureRegulator[1].4		:= iQABPneumatic645_1PressureRegulator1.4;
QABPneumatic645_1PressureRegulator[1].5		:= iQABPneumatic645_1PressureRegulator1.5;
QABPneumatic645_1PressureRegulator[1].6		:= iQABPneumatic645_1PressureRegulator1.6;
QABPneumatic645_1PressureRegulator[1].7		:= iQABPneumatic645_1PressureRegulator1.7;
QABPneumatic645_1PressureRegulator[2].0		:= iQABPneumatic645_1PressureRegulator1.8; 
QABPneumatic645_1PressureRegulator[2].1		:= iQABPneumatic645_1PressureRegulator1.9;                 
QABPneumatic645_1PressureRegulator[2].2		:= iQABPneumatic645_1PressureRegulator1.10;
QABPneumatic645_1PressureRegulator[2].3		:= iQABPneumatic645_1PressureRegulator1.11;
QABPneumatic645_1PressureRegulator[2].4		:= iQABPneumatic645_1PressureRegulator1.12;
QABPneumatic645_1PressureRegulator[2].5		:= iQABPneumatic645_1PressureRegulator1.13;
QABPneumatic645_1PressureRegulator[2].6		:= iQABPneumatic645_1PressureRegulator1.14;
QABPneumatic645_1PressureRegulator[2].7		:= iQABPneumatic645_1PressureRegulator1.15;

IABPneumatic645_1PressureRegulator[1];
IABPneumatic645_1PressureRegulator[2];
iIABPneumatic645_1PressureRegulator1	:= WORD_TO_INT(F_2Bytes_To_Word(byHigh:=IABPneumatic645_1PressureRegulator[2],byLow:=IABPneumatic645_1PressureRegulator[1]));
 

//Zawór proporcjonalny chwytaki pod zakręcarkami szczękowymi
QABPneumatic645_2PressureRegulator[1].0		:= iQABPneumatic645_2PressureRegulator2.0; 
QABPneumatic645_2PressureRegulator[1].1		:= iQABPneumatic645_2PressureRegulator2.1;                 
QABPneumatic645_2PressureRegulator[1].2		:= iQABPneumatic645_2PressureRegulator2.2;
QABPneumatic645_2PressureRegulator[1].3		:= iQABPneumatic645_2PressureRegulator2.3;
QABPneumatic645_2PressureRegulator[1].4		:= iQABPneumatic645_2PressureRegulator2.4;
QABPneumatic645_2PressureRegulator[1].5		:= iQABPneumatic645_2PressureRegulator2.5;
QABPneumatic645_2PressureRegulator[1].6		:= iQABPneumatic645_2PressureRegulator2.6;
QABPneumatic645_2PressureRegulator[1].7		:= iQABPneumatic645_2PressureRegulator2.7;
QABPneumatic645_2PressureRegulator[2].0		:= iQABPneumatic645_2PressureRegulator2.8; 
QABPneumatic645_2PressureRegulator[2].1		:= iQABPneumatic645_2PressureRegulator2.9;                 
QABPneumatic645_2PressureRegulator[2].2		:= iQABPneumatic645_2PressureRegulator2.10;
QABPneumatic645_2PressureRegulator[2].3		:= iQABPneumatic645_2PressureRegulator2.11;
QABPneumatic645_2PressureRegulator[2].4		:= iQABPneumatic645_2PressureRegulator2.12;
QABPneumatic645_2PressureRegulator[2].5		:= iQABPneumatic645_2PressureRegulator2.13;
QABPneumatic645_2PressureRegulator[2].6		:= iQABPneumatic645_2PressureRegulator2.14;
QABPneumatic645_2PressureRegulator[2].7		:= iQABPneumatic645_2PressureRegulator2.15;
                           
IABPneumatic645_2PressureRegulator[1];
IABPneumatic645_2PressureRegulator[2];
iIABPneumatic645_2PressureRegulator1	:= WORD_TO_INT(F_2Bytes_To_Word(byHigh:=IABPneumatic645_2PressureRegulator[2],byLow:=IABPneumatic645_2PressureRegulator[1]));

(*********************Koniec 645 **************************************)
END_ACTION

ACTION aValveCoil:
(*
Nazwa:			aValveCoil
Opis:			Zawory pneumatyczne
Wersja:			v0.1
Data:			2024-10-28
Autor:			DP
Urzadzenia:		
Konfiguracja:	
Info:
*)

//Do podpięcia
P01_TwoPhasesBarriers.QbBarrierBetweenDispencerActuator;	
P01_TwoPhasesBarriers.QbBarrierBetweenWeightActuator;
P01_Gates.QbGate0BeforeDispencersActuator;
P01_Gates.QbGateBeforeDispencersActuator;
P01_Gates.QbLidFeederBarrierActuator;
P01_Gates.QbGateBeforeWeight14Actuator;
P01_Gates.QbGateBeforeWeight56Actuator;
P01_Gates.QbBottleTransferGate1Actuator;
 
P01_BottleFeeder.QbBottleFeederGate1;			
P01_BottleFeeder.QbBottleFeederGate2;					
P01_BottleFeeder.QbBottleFeederArmLeft;			
P01_BottleFeeder.QbBottleFeederArmDown;			
P01_BottleFeeder.QbBottleFeederGripper;			
P01_BottleFeeder.QbBottleFeederFormPositioning;	
P01_BottleFeeder.QbBottleFeederFormGate;			

P01_PucksInserter.QbPucksInserterHammer;
P01_PucksInserter.QbPucksInserterTray;
P01_PucksInserter.QbPucksInserterGate1;
P01_PucksInserter.QbPucksInserterGate2;
P01_PucksInserter.QbPucksInserterFormGate;
P01_PucksInserter.QbPucksInserterFormPositioning;

P02_Dispencers.QbDispencersDragRightDragActuator;
P02_Dispencers.QbDispencersDragLeftDragActuator;
P02_Dispencers.QbDispencersDragLeftLeadBefore1Actuator;
P02_Dispencers.QbDispencersDragLeftLeadAfter1Actuator;
P02_Dispencers.QbDispencersDragRightLeadBefore1Actuator;
P02_Dispencers.QbDispencersDragRightLeadAfter1Actuator;

P02_Dispencers.QbDispencer1SuckingValveActuator;
P02_Dispencers.QbDispencer2SuckingValveActuator;
P02_Dispencers.QbDispencer3SuckingValveActuator;
P02_Dispencers.QbDispencer4SuckingValveActuator;
P02_Dispencers.QbDispencer1DosingValveActuator;
P02_Dispencers.QbDispencer2DosingValveActuator;
P02_Dispencers.QbDispencer3DosingValveActuator;
P02_Dispencers.QbDispencer4DosingValveActuator;
P02_Dispencers.QbDispencersCatch1Actuator;
P02_Dispencers.QbDispencersCatch2Actuator;
P02_Dispencers.QbDispencersCatch3Actuator;
P02_Dispencers.QbDispencersCatch4Actuator;
P02_Dispencers.QbDispencer1DropCatcherValveActuator;
P02_Dispencers.QbDispencer2DropCatcherValveActuator;
P02_Dispencers.QbDispencer3DropCatcherValveActuator;
P02_Dispencers.QbDispencer4DropCatcherValveActuator;
P02_Dispencers.QbDispencersCatchMaxPressure;
P02_Dispencers.QbTank1Pressure;
P02_Dispencers.QbDispencerDropCatcherSuck;

P05_Weight.QbWeight1Actuator;
P05_Weight.QbWeight2Actuator;
P05_Weight.QbWeight3Actuator;
P05_Weight.QbWeight4Actuator;
P05_Weight.QbWeight5Actuator;
P05_Weight.QbWeight6Actuator;

P06_LidFeeder.QbLidFeederDragActuator;
P06_LidFeeder.QbLidFeederDragLeadBefore1Actuator;

P06_LidFeeder.QbLidFeeder_FeederActuator1;
P06_LidFeeder.QbLidFeeder_FeederActuator2;
P06_LidFeeder.QbLidFeeder2_FeederActuator1;
P06_LidFeeder.QbLidFeeder2_FeederActuator2;
P06_LidFeeder.QbLidFeeder2_HeaterActuator;
P06_LidFeeder.QbLidFeeder_HeaterActuator;
P06_LidFeeder.QbLidFeederBlockActuator;
P06_LidFeeder.QbLidFeederFormPositioningActuator; 

P06_LidSealer.QbLidSealer_SealingActuator;
P06_LidSealer.QbLidSealer2_SealingActuator;
P06_LidSealer.QbLidSealerDragActuator;
P06_LidSealer.QbLidSealerBlockActuator;
P06_LidSealer.QbLidSealerDragLeadBefore1Actuator;

P08_CapSorter.QbCapSorterDragActuator;
P08_CapSorter.QbCapSorterDragLeadBefore1Actuator;
P08_CapSorter.QbCapSorterStoperActuator;
QbBlowBeforeGripperScrewer;

QbGateBeforeGripperScrewer;
P10_GripperScrewer.QbGripperScrewersDragActuator;
P10_GripperScrewer.QbGripperScrewersDragLeadBefore1Actuator;
QbGripperScrewerStoperActuator;

P10_GripperScrewer.QbGripperScrewer1Actuator;
P10_GripperScrewer.QbGripperScrewer2Actuator;
P10_GripperScrewer.QbGripperScrewer1CatchActuator;
P10_GripperScrewer.QbGripperScrewer2CatchActuator;

		
(*************************** 641 **************************************)
QABPneumatic641ValveCoils[1].0	:= P02_Dispencers.QbDispencer1SuckingValveActuator;			//Siłownik:	zawór ssący 1		
QABPneumatic641ValveCoils[1].1	;											                           	                
QABPneumatic641ValveCoils[1].2	:= P02_Dispencers.QbDispencer2SuckingValveActuator;  		//Siłownik:	zawór ssący 2	
QABPneumatic641ValveCoils[1].3	; 										                               	           
QABPneumatic641ValveCoils[1].4	:= P02_Dispencers.QbDispencer3SuckingValveActuator;			//Siłownik:	zawór ssący 3		
QABPneumatic641ValveCoils[1].5	;									                                   	          
QABPneumatic641ValveCoils[1].6	:= P02_Dispencers.QbDispencer4SuckingValveActuator;			//Siłownik:	zawór ssący 4		
QABPneumatic641ValveCoils[1].7	;								

QABPneumatic641ValveCoils[2].0	:=	P02_Dispencers.QbDispencer1DosingValveActuator;			//Siłownik: zawór tłoczący 1 
QABPneumatic641ValveCoils[2].1	:=	NOT P02_Dispencers.QbDispencer1DosingValveActuator;                        
QABPneumatic641ValveCoils[2].2	:=	P02_Dispencers.QbDispencer2DosingValveActuator;			//Siłownik: zawór tłoczący 2 
QABPneumatic641ValveCoils[2].3	:=	NOT P02_Dispencers.QbDispencer2DosingValveActuator;                         
QABPneumatic641ValveCoils[2].4	:=	P02_Dispencers.QbDispencer3DosingValveActuator;			//Siłownik: zawór tłoczący 3
QABPneumatic641ValveCoils[2].5	:=	NOT P02_Dispencers.QbDispencer3DosingValveActuator;	                         
QABPneumatic641ValveCoils[2].6	:=  P02_Dispencers.QbDispencer4DosingValveActuator;			//Siłownik: zawór tłoczący 4
QABPneumatic641ValveCoils[2].7	:=	NOT P02_Dispencers.QbDispencer4DosingValveActuator ;                 

QABPneumatic641ValveCoils[3].0	:= P02_Dispencers.QbDispencer1DropCatcherValveActuator;		//Siłownik:	tacka ociekowa 1    
QABPneumatic641ValveCoils[3].1	;	                                                                   	                   
QABPneumatic641ValveCoils[3].2	:= P02_Dispencers.QbDispencer2DropCatcherValveActuator;		//Siłownik:	tacka ociekowa 2   
QABPneumatic641ValveCoils[3].3	;			                                                           	                         
QABPneumatic641ValveCoils[3].4	:= P02_Dispencers.QbDispencer3DropCatcherValveActuator;		//Siłownik:	tacka ociekowa 3	   
QABPneumatic641ValveCoils[3].5	;                                                                      	                 
QABPneumatic641ValveCoils[3].6	:= P02_Dispencers.QbDispencer4DropCatcherValveActuator; 	//Siłownik:	tacka ociekowa 4 
QABPneumatic641ValveCoils[3].7	;		                                                                                     

QABPneumatic641ValveCoils[4].0	:= P02_Dispencers.QbTank1Pressure	; //Nadciśnienie w zbiorniku masy  
QABPneumatic641ValveCoils[4].1	; //rezerwa
QABPneumatic641ValveCoils[4].2	:= NOT P02_Dispencers.QbDispencersCatch2Actuator;  
QABPneumatic641ValveCoils[4].3	:= NOT P02_Dispencers.QbDispencersCatch1Actuator;  
QABPneumatic641ValveCoils[4].4	:= NOT P02_Dispencers.QbDispencersCatch4Actuator;  
QABPneumatic641ValveCoils[4].5	:= NOT P02_Dispencers.QbDispencersCatch3Actuator;  
QABPneumatic641ValveCoils[4].6	;     
QABPneumatic641ValveCoils[4].7	;		    
                                
QABPneumatic641ValveCoils[5].0	:=  P02_Dispencers.QbDispencersCatch2Actuator;			//Siłownik: centrowanie szyjki 1	  
QABPneumatic641ValveCoils[5].1	:=  P02_Dispencers.QbDispencersCatch1Actuator;                                        
QABPneumatic641ValveCoils[5].2	:=  P02_Dispencers.QbDispencersCatch4Actuator; 				  
QABPneumatic641ValveCoils[5].3	:=  P02_Dispencers.QbDispencersCatch3Actuator;                  
QABPneumatic641ValveCoils[5].4	;				 
QABPneumatic641ValveCoils[5].5	;                   
QABPneumatic641ValveCoils[5].6	;					  
QABPneumatic641ValveCoils[5].7	; 

QABPneumatic641ValveCoils[6].0	;
QABPneumatic641ValveCoils[6].1	;
QABPneumatic641ValveCoils[6].2	;
QABPneumatic641ValveCoils[6].3	;
QABPneumatic641ValveCoils[6].4	;
QABPneumatic641ValveCoils[6].5	;
QABPneumatic641ValveCoils[6].6	;
QABPneumatic641ValveCoils[6].7	;

(***************************Koniec 641 **************************************)

(*************************** 642 **************************************)
QABPneumatic642ValveCoils[1].0	:= NOT p01_twophasesbarriers.QbBarrierBetweenDispencerActuator;
QABPneumatic642ValveCoils[1].1	:= 	   p01_twophasesbarriers.QbBarrierBetweenDispencerActuator; 
QABPneumatic642ValveCoils[1].2	:= NOT P01_TwoPhasesBarriers.QbBarrierBetweenWeightActuator;
QABPneumatic642ValveCoils[1].3	:=  P01_TwoPhasesBarriers.QbBarrierBetweenWeightActuator;
QABPneumatic642ValveCoils[1].4	:=     P02_Dispencers.QbDispencersDragLeftDragActuator;	
QABPneumatic642ValveCoils[1].5	:= NOT P02_Dispencers.QbDispencersDragLeftDragActuator;  
QABPneumatic642ValveCoils[1].6	:=     P02_Dispencers.QbDispencersDragRightDragActuator;		      
QABPneumatic642ValveCoils[1].7	:= NOT P02_Dispencers.QbDispencersDragRightDragActuator;		   		
                                        
QABPneumatic642ValveCoils[2].0	:=	   P02_Dispencers.QbDispencersDragLeftLeadBefore1Actuator;			  
QABPneumatic642ValveCoils[2].1	:= NOT P02_Dispencers.QbDispencersDragLeftLeadBefore1Actuator;  	            		
QABPneumatic642ValveCoils[2].2	:=	   P02_Dispencers.QbDispencersDragRightLeadBefore1Actuator;	
QABPneumatic642ValveCoils[2].3	:= NOT P02_Dispencers.QbDispencersDragRightLeadBefore1Actuator; 
QABPneumatic642ValveCoils[2].4	:=     P01_Gates.QbGate0BeforeDispencersActuator; 	//szlaban przed dozownikami wcześniejszy
QABPneumatic642ValveCoils[2].5	:= NOT P01_Gates.QbGate0BeforeDispencersActuator;  	
QABPneumatic642ValveCoils[2].6	:=		P01_Gates.QbGate0BeforeDispencersActuator;   ////szlaban przed dozownikami późniejszy              
QABPneumatic642ValveCoils[2].7	:=  NOT P01_Gates.QbGate0BeforeDispencersActuator;	           		
                                       
QABPneumatic642ValveCoils[3].0	:=   p01_gates.QbBottleTransferGate1Actuator;              
QABPneumatic642ValveCoils[3].1	:=  NOT p01_gates.QbBottleTransferGate1Actuator; 			
QABPneumatic642ValveCoils[3].2	:=   QbBlowAfterGripperScrewer;                 
QABPneumatic642ValveCoils[3].3	:=     P02_Dispencers.QbDispencerDropCatcherSuck;    
QABPneumatic642ValveCoils[3].4	;
QABPneumatic642ValveCoils[3].5	;
QABPneumatic642ValveCoils[3].6	;
QABPneumatic642ValveCoils[3].7	;
 
QABPneumatic642ValveCoils[4].0		; 
QABPneumatic642ValveCoils[4].1		; 
QABPneumatic642ValveCoils[4].2		; 
QABPneumatic642ValveCoils[4].3		; 
QABPneumatic642ValveCoils[4].4		; 
QABPneumatic642ValveCoils[4].5		; 
QABPneumatic642ValveCoils[4].6		; 
QABPneumatic642ValveCoils[4].7		;
 
QABPneumatic642ValveCoils[5].0		; 
QABPneumatic642ValveCoils[5].1		; 
QABPneumatic642ValveCoils[5].2		; 
QABPneumatic642ValveCoils[5].3		; 
QABPneumatic642ValveCoils[5].4		; 
QABPneumatic642ValveCoils[5].5		; 
QABPneumatic642ValveCoils[5].6		; 
QABPneumatic642ValveCoils[5].7		; 
(***************************Koniec 642 **************************************)

(*************************** 643 **************************************)
QABPneumatic643ValveCoils[1].0		:=	P05_Weight.QbWeight1Actuator;//QbWeight1ActuatorUp;			     :=  
QABPneumatic643ValveCoils[1].1		:=	NOT P05_Weight.QbWeight1Actuator;//QbWeight1ActuatorDown;        :=  
QABPneumatic643ValveCoils[1].2		:= 	P05_Weight.QbWeight2Actuator;//QbWeight2ActuatorUp; 		     :=  
QABPneumatic643ValveCoils[1].3		:= 	NOT P05_Weight.QbWeight2Actuator;//QbWeight2ActuatorDown;        := 
QABPneumatic643ValveCoils[1].4		:= 	P05_Weight.QbWeight3Actuator;//QbWeight3ActuatorUp; 		     := 
QABPneumatic643ValveCoils[1].5		:=  NOT P05_Weight.QbWeight3Actuator;//QbWeight3ActuatorDown;        := 
QABPneumatic643ValveCoils[1].6		:= 	P05_Weight.QbWeight4Actuator;//QbWeight4ActuatorUp;		         :=  
QABPneumatic643ValveCoils[1].7		:=  NOT P05_Weight.QbWeight4Actuator;//QbWeight4ActuatorDown;        :=  
                                                                                                         
QABPneumatic643ValveCoils[2].0		:=  P05_Weight.QbWeight5Actuator; 			                                       
QABPneumatic643ValveCoils[2].1		:=  NOT P05_Weight.QbWeight5Actuator;  			                                          
QABPneumatic643ValveCoils[2].2		:=  P05_Weight.QbWeight6Actuator; 		                                       
QABPneumatic643ValveCoils[2].3		:=  NOT P05_Weight.QbWeight6Actuator; 		                                          
QABPneumatic643ValveCoils[2].4		:= P01_Gates.QbGateBeforeWeight14Actuator;						                                                           
QABPneumatic643ValveCoils[2].5		:= NOT P01_Gates.QbGateBeforeWeight14Actuator;                                                               
QABPneumatic643ValveCoils[2].6		:= P01_gates.QbGateBeforeWeight56Actuator;						                                                           
QABPneumatic643ValveCoils[2].7		:= NOT P01_gates.QbGateBeforeWeight56Actuator;				                                                  
                                                                                                    
QABPneumatic643ValveCoils[3].0		:= P02_Dispencers.QbDispencersDragLeftLeadAfter1Actuator;		                                                         
QABPneumatic643ValveCoils[3].1		:= NOT P02_Dispencers.QbDispencersDragLeftLeadAfter1Actuator;	                                                           
QABPneumatic643ValveCoils[3].2		:= P02_Dispencers.QbDispencersDragrightLeadAfter1Actuator;		
QABPneumatic643ValveCoils[3].3		:= NOT P02_Dispencers.QbDispencersDragrightLeadAfter1Actuator;	
QABPneumatic643ValveCoils[3].4		; 
QABPneumatic643ValveCoils[3].5		; 
QABPneumatic643ValveCoils[3].6		; 
QABPneumatic643ValveCoils[3].7		;

QABPneumatic643ValveCoils[4].0		; 
QABPneumatic643ValveCoils[4].1		; 
QABPneumatic643ValveCoils[4].2		; 
QABPneumatic643ValveCoils[4].3		; 
QABPneumatic643ValveCoils[4].4		; 
QABPneumatic643ValveCoils[4].5		; 
QABPneumatic643ValveCoils[4].6		; 
QABPneumatic643ValveCoils[4].7		;
 
QABPneumatic643ValveCoils[5].0		; 
QABPneumatic643ValveCoils[5].1		; 
QABPneumatic643ValveCoils[5].2		; 
QABPneumatic643ValveCoils[5].3		; 
QABPneumatic643ValveCoils[5].4		; 
QABPneumatic643ValveCoils[5].5		; 
QABPneumatic643ValveCoils[5].6		; 
QABPneumatic643ValveCoils[5].7		; 
(***************************Koniec 643 **************************************)

(*************************** 644 **************************************)
QABPneumatic644ValveCoils[1].0		:=	P01_Gates.QbLidFeederBarrierActuator;
QABPneumatic644ValveCoils[1].1		:= NOT P01_Gates.QbLidFeederBarrierActuator;
QABPneumatic644ValveCoils[1].2		:= P06_WickFeeder.QbFormPositioning;
QABPneumatic644ValveCoils[1].3		:=FALSE;
QABPneumatic644ValveCoils[1].4		:= P06_WickFeeder.QbWickFeederDragLeadBefore1Actuator;  			
QABPneumatic644ValveCoils[1].5		:= NOT P06_WickFeeder.QbWickFeederDragLeadBefore1Actuator;  									
QABPneumatic644ValveCoils[1].6		:= P06_WickFeeder.QbWickFeederDragActuator;	                  
QABPneumatic644ValveCoils[1].7		:= NOT P06_WickFeeder.QbWickFeederDragActuator;	 	
                                            	
QABPneumatic644ValveCoils[2].0		:= P06_LidSealer.QbLidSealerDragLeadBefore1Actuator;	
QABPneumatic644ValveCoils[2].1		:= NOT P06_LidSealer.QbLidSealerDragLeadBefore1Actuator;		
QABPneumatic644ValveCoils[2].2		:=P06_LidSealer.QbLidSealerDragActuator;
QABPneumatic644ValveCoils[2].3		:= NOT P06_LidSealer.QbLidSealerDragActuator;
QABPneumatic644ValveCoils[2].4		:= P10_GripperScrewer.QbGripperScrewersDragLeadBefore1Actuator; 	  
QABPneumatic644ValveCoils[2].5		:= NOT P10_GripperScrewer.QbGripperScrewersDragLeadBefore1Actuator; 
QABPneumatic644ValveCoils[2].6		:= P10_GripperScrewer.QbGripperScrewersDragActuator;		 
QABPneumatic644ValveCoils[2].7		:= NOT P10_GripperScrewer.QbGripperScrewersDragActuator; 

QABPneumatic644ValveCoils[3].0		; //rezerwa
QABPneumatic644ValveCoils[3].1		; //rezerwa
QABPneumatic644ValveCoils[3].2		; //rezerwa
QABPneumatic644ValveCoils[3].3		; //rezerwa
QABPneumatic644ValveCoils[3].4		:= QbGripperScrewerAcceleratorActuator;
QABPneumatic644ValveCoils[3].5		:=FALSE;
QABPneumatic644ValveCoils[3].6		:= QbGripperScrewerStoperActuator;
QABPneumatic644ValveCoils[3].7		:=FALSE;
 
QABPneumatic644ValveCoils[4].0		:=P06_LidSealer.QbLidSealerStoperActuatorOn;
QABPneumatic644ValveCoils[4].1		:=FALSE; 
QABPneumatic644ValveCoils[4].2		; 
QABPneumatic644ValveCoils[4].3		; 
QABPneumatic644ValveCoils[4].4		; 
QABPneumatic644ValveCoils[4].5		; 
QABPneumatic644ValveCoils[4].6		; 
QABPneumatic644ValveCoils[4].7		;
 
QABPneumatic644ValveCoils[5].0		; 
QABPneumatic644ValveCoils[5].1		; 
QABPneumatic644ValveCoils[5].2		; 
QABPneumatic644ValveCoils[5].3		; 
QABPneumatic644ValveCoils[5].4		; 
QABPneumatic644ValveCoils[5].5		; 
QABPneumatic644ValveCoils[5].6		; 
QABPneumatic644ValveCoils[5].7		; 
(***************************Koniec 644 **************************************)

(*************************** 645 **************************************)
QABPneumatic645ValveCoils[1].0		:= P10_GripperScrewer.QbGripperScrewer2Actuator; 		
QABPneumatic645ValveCoils[1].1		:= P10_GripperScrewer.QbGripperScrewer1Actuator;		
QABPneumatic645ValveCoils[1].2		:= P10_GripperScrewer.QbGripperScrewer1CatchActuator;
QABPneumatic645ValveCoils[1].3		:= FALSE;                                            
QABPneumatic645ValveCoils[1].4		:= P10_GripperScrewer.QbGripperScrewer2CatchActuator;
QABPneumatic645ValveCoils[1].5		:= FALSE;                                            
QABPneumatic645ValveCoils[1].6		; 
QABPneumatic645ValveCoils[1].7		;
              
QABPneumatic645ValveCoils[2].0		; 
QABPneumatic645ValveCoils[2].1		; 
QABPneumatic645ValveCoils[2].2		; 
QABPneumatic645ValveCoils[2].3		; 
QABPneumatic645ValveCoils[2].4		; 
QABPneumatic645ValveCoils[2].5		; 
QABPneumatic645ValveCoils[2].6		; 
QABPneumatic645ValveCoils[2].7		;
(***************************Koniec 645 **************************************)

(*************************** 646 **************************************)
//Platynki
(*QABPneumatic646ValveCoils[1].0		:= P06_LidFeeder.QbLidFeeder2_FeederActuator1	;	//pobieranie i ruch w dół 						
QABPneumatic646ValveCoils[1].1		:= NOT P06_LidFeeder.QbLidFeeder2_FeederActuator1;    //pobieranie i ruch w dół                        
QABPneumatic646ValveCoils[1].2		:= P06_LidFeeder.QbLidFeeder2_FeederActuator2;		//wbicie wkładki       
QABPneumatic646ValveCoils[1].3		:= NOT P06_LidFeeder.QbLidFeeder2_FeederActuator2; 	//wbicie wkładki         
QABPneumatic646ValveCoils[1].4		:= P06_LidFeeder.QbLidFeeder_FeederActuator1	;	    //pobieranie wkładki 2                          
QABPneumatic646ValveCoils[1].5		:= NOT P06_LidFeeder.QbLidFeeder_FeederActuator1;  //pobieranie wkładki 2                              
QABPneumatic646ValveCoils[1].6		:= P06_LidFeeder.QbLidFeeder_FeederActuator2;		    //odkładanie wkładki 2                          
QABPneumatic646ValveCoils[1].7		:= NOT P06_LidFeeder.QbLidFeeder_FeederActuator2;  //odkładanie wkładki 2                              
                                                                                                
QABPneumatic646ValveCoils[2].0		;                                                          
QABPneumatic646ValveCoils[2].1		;                                                          
QABPneumatic646ValveCoils[2].2		;                                                          
QABPneumatic646ValveCoils[2].3		;                                                           
QABPneumatic646ValveCoils[2].4		;                                                           
QABPneumatic646ValveCoils[2].5		; 
QABPneumatic646ValveCoils[2].6		; 
QABPneumatic646ValveCoils[2].7		;
 
QABPneumatic646ValveCoils[3].0		:= P06_LidFeeder.QbLidFeeder_SuckerActuator ;
QABPneumatic646ValveCoils[3].1		:= P06_LidFeeder.QbLidFeeder2_SuckerActuator  ;*)
//Knoty
QABPneumatic646ValveCoils[1].0		:= NOT P06_WickFeeder.QbStopper1;	// u góry			           
QABPneumatic646ValveCoils[1].1		:= NOT P06_WickFeeder.QbStopper2;              
QABPneumatic646ValveCoils[1].2		:= P06_WickFeeder.QbSeparator1;			            
QABPneumatic646ValveCoils[1].3		:= P06_WickFeeder.QbSeparator2	;		         
QABPneumatic646ValveCoils[1].4		:= P06_WickFeeder.QbSleve1SeparatorActOut	;            
QABPneumatic646ValveCoils[1].5		:= P06_WickFeeder.QbSleve1SeparatorActIn	;                  
QABPneumatic646ValveCoils[1].6		:= P06_WickFeeder.QbSleve2SeparatorActOut	;                  
QABPneumatic646ValveCoils[1].7		:= P06_WickFeeder.QbSleve2SeparatorActIn	;                                                                 	           
QABPneumatic646ValveCoils[2].0		:=	P06_WickFeeder.QbHammer1;	            
QABPneumatic646ValveCoils[2].1		:=	NOT P06_WickFeeder.QbHammer1;	      ;     
QABPneumatic646ValveCoils[2].2		:= 	P06_WickFeeder.QbHammer2			      ; 
QABPneumatic646ValveCoils[2].3		:=  NOT P06_WickFeeder.QbHammer2			 		  ;
QABPneumatic646ValveCoils[2].4		:=  P06_WickFeeder.QbBlow1	;		
QABPneumatic646ValveCoils[2].5		:= P06_WickFeeder.QbSleeveBlow;			
QABPneumatic646ValveCoils[2].6		;
QABPneumatic646ValveCoils[2].7		;
                                    
QABPneumatic646ValveCoils[3].0		;
QABPneumatic646ValveCoils[3].1		;
(***************************Koniec 646 **************************************)

